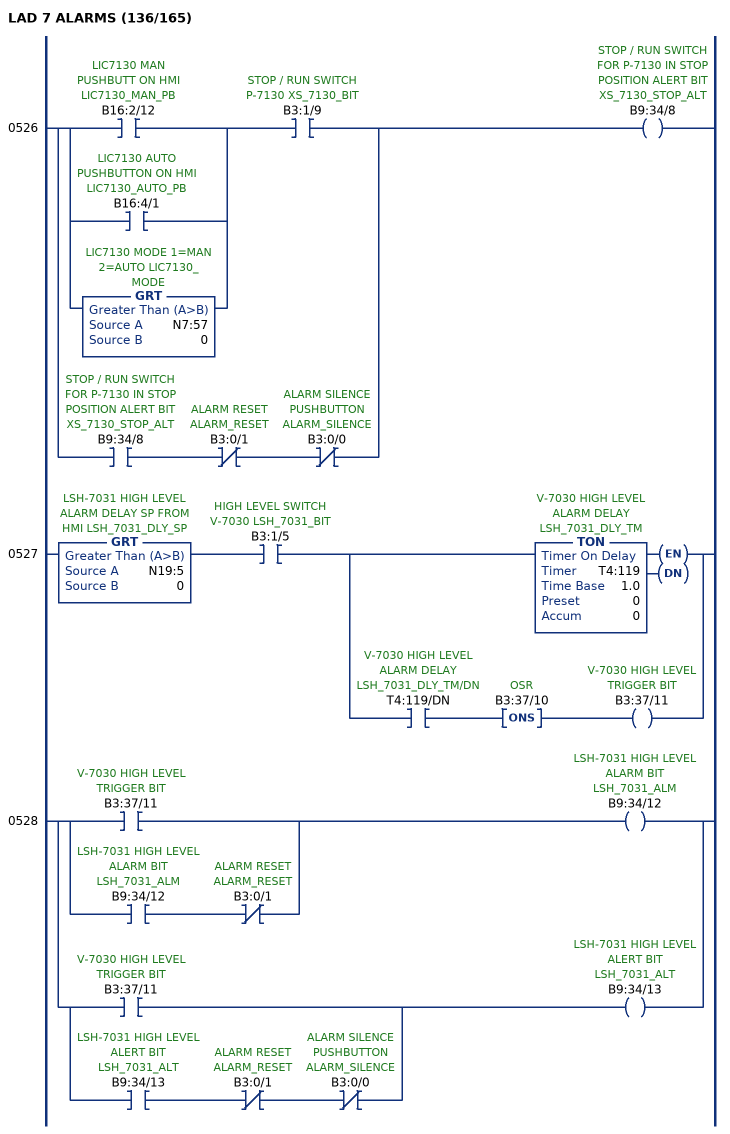
% Rung: 526 %
SOR BST BST XIC B16:2/12 NXB XIC B16:4/1 NXB GRT N7:57 0 BND XIC B3:1/9 NXB XIC B9:34/8 XIO B3:0/1 XIO B3:0/0 BND OTE B9:34/8 EOR
%   B16:2/12  LIC7130_MAN_PB  "LIC7130 MAN PUSHBUTT ON HMI" %
%   B16:4/1  LIC7130_AUTO_PB  "LIC7130 AUTO PUSHBUTTON ON HMI" %
%   N7:57  LIC7130_MODE  "LIC7130 MODE 1=MAN 2=AUTO" %
%   B3:1/9  XS_7130_BIT  "STOP / RUN SWITCH P-7130" %
%   B9:34/8  XS_7130_STOP_ALT  "STOP / RUN SWITCH FOR P-7130 IN STOP POSITION ALERT BIT" %
%   B3:0/1  ALARM_RESET  "ALARM RESET" %
%   B3:0/0  ALARM_SILENCE  "ALARM SILENCE PUSHBUTTON" %
% Rung: 527 %
SOR GRT N19:5 0 XIC B3:1/5 BST TON T4:119 1.0 0 0 NXB XIC T4:119/DN OSR B3:37/10 OTE B3:37/11 BND EOR
%   N19:5  LSH_7031_DLY_SP  "LSH-7031 HIGH LEVEL ALARM DELAY SP FROM HMI" %
%   B3:1/5  LSH_7031_BIT  "HIGH LEVEL SWITCH V-7030" %
%   T4:119  LSH_7031_DLY_TM  "V-7030 HIGH LEVEL ALARM DELAY" %
%   B3:37/10  "OSR" %
%   B3:37/11  "V-7030 HIGH LEVEL TRIGGER BIT" %
% Rung: 528 %
SOR BST BST XIC B3:37/11 NXB XIC B9:34/12 XIO B3:0/1 BND OTE B9:34/12 NXB BST XIC B3:37/11 NXB XIC B9:34/13 XIO B3:0/1 XIO B3:0/0 BND OTE B9:34/13 BND EOR
%   B3:37/11  "V-7030 HIGH LEVEL TRIGGER BIT" %
%   B9:34/12  LSH_7031_ALM  "LSH-7031 HIGH LEVEL ALARM BIT" %
%   B3:0/1  ALARM_RESET  "ALARM RESET" %
%   B9:34/13  LSH_7031_ALT  "LSH-7031 HIGH LEVEL ALERT BIT" %
%   B3:0/0  ALARM_SILENCE  "ALARM SILENCE PUSHBUTTON" %

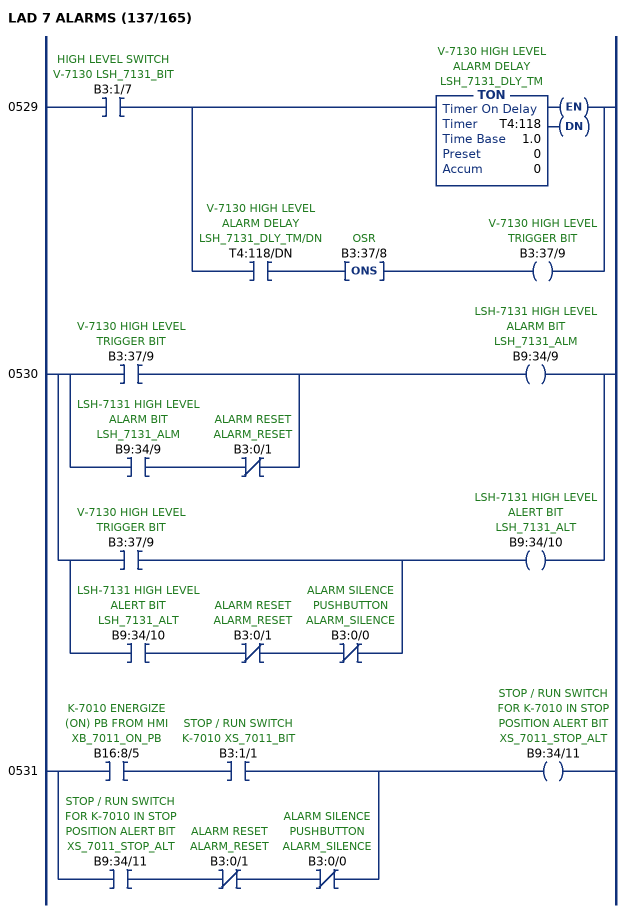
% Rung: 529 %
SOR XIC B3:1/7 BST TON T4:118 1.0 0 0 NXB XIC T4:118/DN OSR B3:37/8 OTE B3:37/9 BND EOR
%   B3:1/7  LSH_7131_BIT  "HIGH LEVEL SWITCH V-7130" %
%   T4:118  LSH_7131_DLY_TM  "V-7130 HIGH LEVEL ALARM DELAY" %
%   B3:37/8  "OSR" %
%   B3:37/9  "V-7130 HIGH LEVEL TRIGGER BIT" %
% Rung: 530 %
SOR BST BST XIC B3:37/9 NXB XIC B9:34/9 XIO B3:0/1 BND OTE B9:34/9 NXB BST XIC B3:37/9 NXB XIC B9:34/10 XIO B3:0/1 XIO B3:0/0 BND OTE B9:34/10 BND EOR
%   B3:37/9  "V-7130 HIGH LEVEL TRIGGER BIT" %
%   B9:34/9  LSH_7131_ALM  "LSH-7131 HIGH LEVEL ALARM BIT" %
%   B3:0/1  ALARM_RESET  "ALARM RESET" %
%   B9:34/10  LSH_7131_ALT  "LSH-7131 HIGH LEVEL ALERT BIT" %
%   B3:0/0  ALARM_SILENCE  "ALARM SILENCE PUSHBUTTON" %
% Rung: 531 %
SOR BST XIC B16:8/5 XIC B3:1/1 NXB XIC B9:34/11 XIO B3:0/1 XIO B3:0/0 BND OTE B9:34/11 EOR
%   B16:8/5  XB_7011_ON_PB  "K-7010 ENERGIZE (ON) PB FROM HMI" %
%   B3:1/1  XS_7011_BIT  "STOP / RUN SWITCH K-7010" %
%   B9:34/11  XS_7011_STOP_ALT  "STOP / RUN SWITCH FOR K-7010 IN STOP POSITION ALERT BIT" %
%   B3:0/1  ALARM_RESET  "ALARM RESET" %
%   B3:0/0  ALARM_SILENCE  "ALARM SILENCE PUSHBUTTON" %

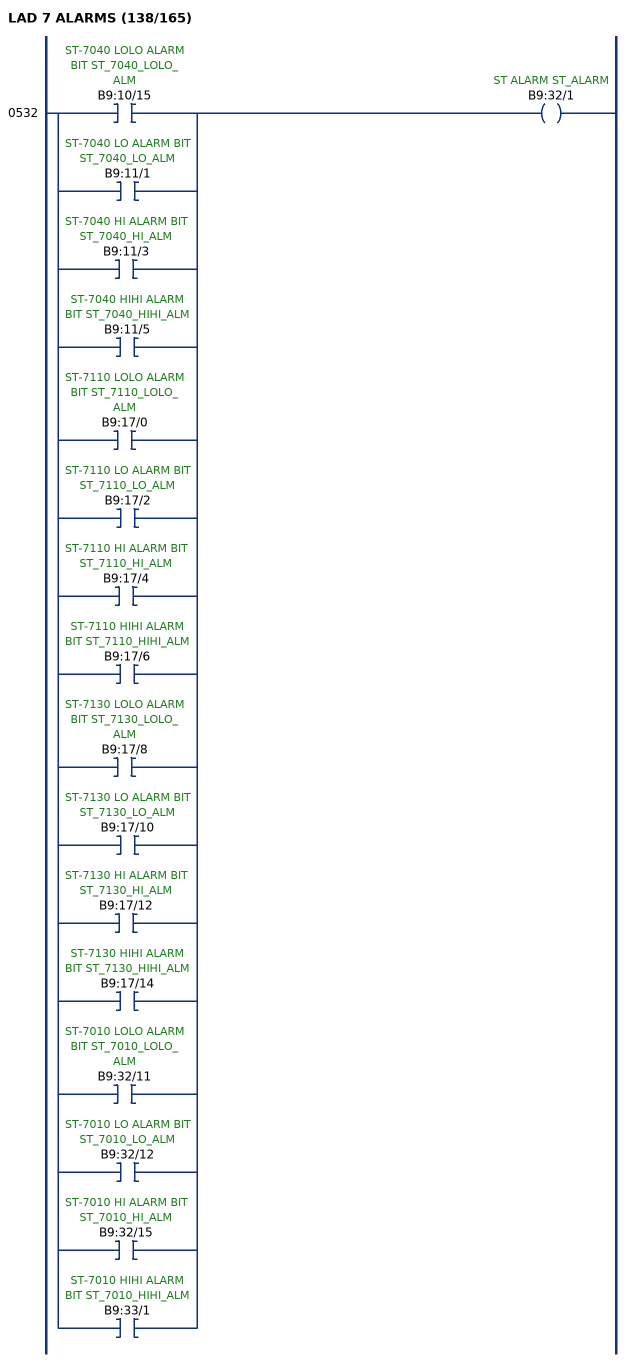
% Rung: 532 %
SOR BST XIC B9:10/15 NXB XIC B9:11/1 NXB XIC B9:11/3 NXB XIC B9:11/5 NXB XIC B9:17/0 NXB XIC B9:17/2 NXB XIC B9:17/4 NXB XIC B9:17/6 NXB XIC B9:17/8 NXB XIC B9:17/10 NXB XIC B9:17/12 NXB XIC B9:17/14 NXB XIC B9:32/11 NXB XIC B9:32/12 NXB XIC B9:32/15 NXB XIC B9:33/1 BND OTE B9:32/1 EOR
%   B9:10/15  ST_7040_LOLO_ALM  "ST-7040 LOLO ALARM BIT" %
%   B9:11/1  ST_7040_LO_ALM  "ST-7040 LO ALARM BIT" %
%   B9:11/3  ST_7040_HI_ALM  "ST-7040 HI ALARM BIT" %
%   B9:11/5  ST_7040_HIHI_ALM  "ST-7040 HIHI ALARM BIT" %
%   B9:17/0  ST_7110_LOLO_ALM  "ST-7110 LOLO ALARM BIT" %
%   B9:17/2  ST_7110_LO_ALM  "ST-7110 LO ALARM BIT" %
%   B9:17/4  ST_7110_HI_ALM  "ST-7110 HI ALARM BIT" %
%   B9:17/6  ST_7110_HIHI_ALM  "ST-7110 HIHI ALARM BIT" %
%   B9:17/8  ST_7130_LOLO_ALM  "ST-7130 LOLO ALARM BIT" %
%   B9:17/10  ST_7130_LO_ALM  "ST-7130 LO ALARM BIT" %
%   B9:17/12  ST_7130_HI_ALM  "ST-7130 HI ALARM BIT" %
%   B9:17/14  ST_7130_HIHI_ALM  "ST-7130 HIHI ALARM BIT" %
%   B9:32/11  ST_7010_LOLO_ALM  "ST-7010 LOLO ALARM BIT" %
%   B9:32/12  ST_7010_LO_ALM  "ST-7010 LO ALARM BIT" %
%   B9:32/15  ST_7010_HI_ALM  "ST-7010 HI ALARM BIT" %
%   B9:33/1  ST_7010_HIHI_ALM  "ST-7010 HIHI ALARM BIT" %
%   B9:32/1  ST_ALARM  "ST ALARM" %

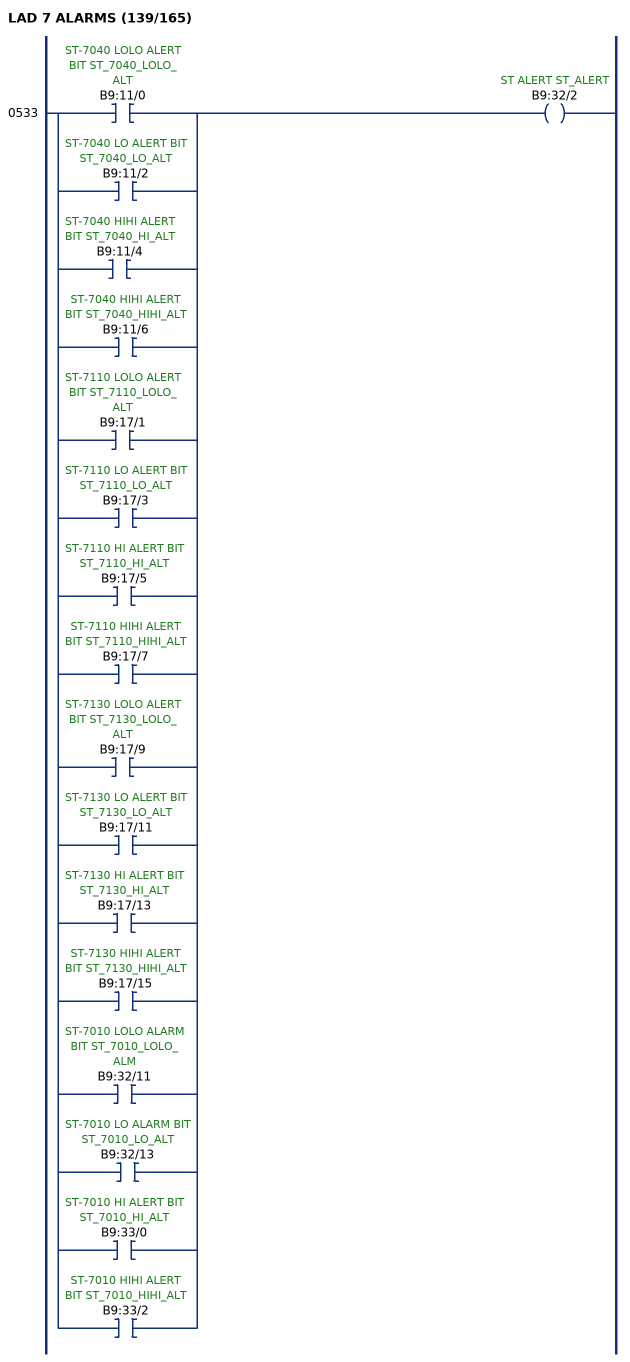
% Rung: 533 %
SOR BST XIC B9:11/0 NXB XIC B9:11/2 NXB XIC B9:11/4 NXB XIC B9:11/6 NXB XIC B9:17/1 NXB XIC B9:17/3 NXB XIC B9:17/5 NXB XIC B9:17/7 NXB XIC B9:17/9 NXB XIC B9:17/11 NXB XIC B9:17/13 NXB XIC B9:17/15 NXB XIC B9:32/11 NXB XIC B9:32/13 NXB XIC B9:33/0 NXB XIC B9:33/2 BND OTE B9:32/2 EOR
%   B9:11/0  ST_7040_LOLO_ALT  "ST-7040 LOLO ALERT BIT" %
%   B9:11/2  ST_7040_LO_ALT  "ST-7040 LO ALERT BIT" %
%   B9:11/4  ST_7040_HI_ALT  "ST-7040 HIHI ALERT BIT" %
%   B9:11/6  ST_7040_HIHI_ALT  "ST-7040 HIHI ALERT BIT" %
%   B9:17/1  ST_7110_LOLO_ALT  "ST-7110 LOLO ALERT BIT" %
%   B9:17/3  ST_7110_LO_ALT  "ST-7110 LO ALERT BIT" %
%   B9:17/5  ST_7110_HI_ALT  "ST-7110 HI ALERT BIT" %
%   B9:17/7  ST_7110_HIHI_ALT  "ST-7110 HIHI ALERT BIT" %
%   B9:17/9  ST_7130_LOLO_ALT  "ST-7130 LOLO ALERT BIT" %
%   B9:17/11  ST_7130_LO_ALT  "ST-7130 LO ALERT BIT" %
%   B9:17/13  ST_7130_HI_ALT  "ST-7130 HI ALERT BIT" %
%   B9:17/15  ST_7130_HIHI_ALT  "ST-7130 HIHI ALERT BIT" %
%   B9:32/11  ST_7010_LOLO_ALM  "ST-7010 LOLO ALARM BIT" %
%   B9:32/13  ST_7010_LO_ALT  "ST-7010 LO ALARM BIT" %
%   B9:33/0  ST_7010_HI_ALT  "ST-7010 HI ALERT BIT" %
%   B9:33/2  ST_7010_HIHI_ALT  "ST-7010 HIHI ALERT BIT" %
%   B9:32/2  ST_ALERT  "ST ALERT" %

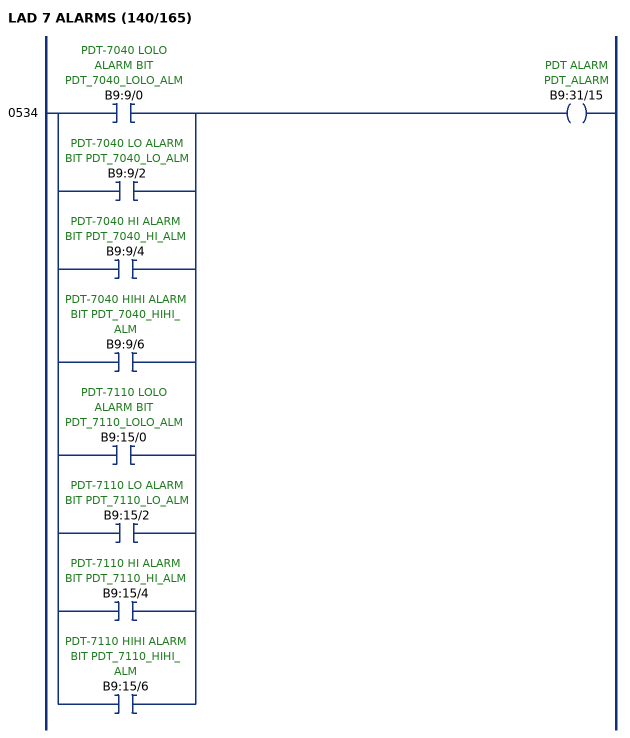
% Rung: 534 %
SOR BST XIC B9:9/0 NXB XIC B9:9/2 NXB XIC B9:9/4 NXB XIC B9:9/6 NXB XIC B9:15/0 NXB XIC B9:15/2 NXB XIC B9:15/4 NXB XIC B9:15/6 BND OTE B9:31/15 EOR
%   B9:9/0  PDT_7040_LOLO_ALM  "PDT-7040 LOLO ALARM BIT" %
%   B9:9/2  PDT_7040_LO_ALM  "PDT-7040 LO ALARM BIT" %
%   B9:9/4  PDT_7040_HI_ALM  "PDT-7040 HI ALARM BIT" %
%   B9:9/6  PDT_7040_HIHI_ALM  "PDT-7040 HIHI ALARM BIT" %
%   B9:15/0  PDT_7110_LOLO_ALM  "PDT-7110 LOLO ALARM BIT" %
%   B9:15/2  PDT_7110_LO_ALM  "PDT-7110 LO ALARM BIT" %
%   B9:15/4  PDT_7110_HI_ALM  "PDT-7110 HI ALARM BIT" %
%   B9:15/6  PDT_7110_HIHI_ALM  "PDT-7110 HIHI ALARM BIT" %
%   B9:31/15  PDT_ALARM  "PDT ALARM" %

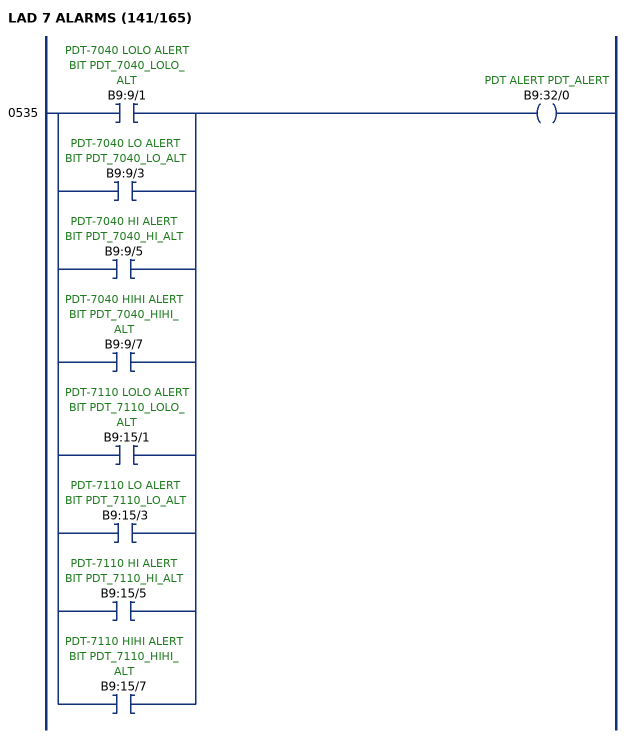
% Rung: 535 %
SOR BST XIC B9:9/1 NXB XIC B9:9/3 NXB XIC B9:9/5 NXB XIC B9:9/7 NXB XIC B9:15/1 NXB XIC B9:15/3 NXB XIC B9:15/5 NXB XIC B9:15/7 BND OTE B9:32/0 EOR
%   B9:9/1  PDT_7040_LOLO_ALT  "PDT-7040 LOLO ALERT BIT" %
%   B9:9/3  PDT_7040_LO_ALT  "PDT-7040 LO ALERT BIT" %
%   B9:9/5  PDT_7040_HI_ALT  "PDT-7040 HI ALERT BIT" %
%   B9:9/7  PDT_7040_HIHI_ALT  "PDT-7040 HIHI ALERT BIT" %
%   B9:15/1  PDT_7110_LOLO_ALT  "PDT-7110 LOLO ALERT BIT" %
%   B9:15/3  PDT_7110_LO_ALT  "PDT-7110 LO ALERT BIT" %
%   B9:15/5  PDT_7110_HI_ALT  "PDT-7110 HI ALERT BIT" %
%   B9:15/7  PDT_7110_HIHI_ALT  "PDT-7110 HIHI ALERT BIT" %
%   B9:32/0  PDT_ALERT  "PDT ALERT" %

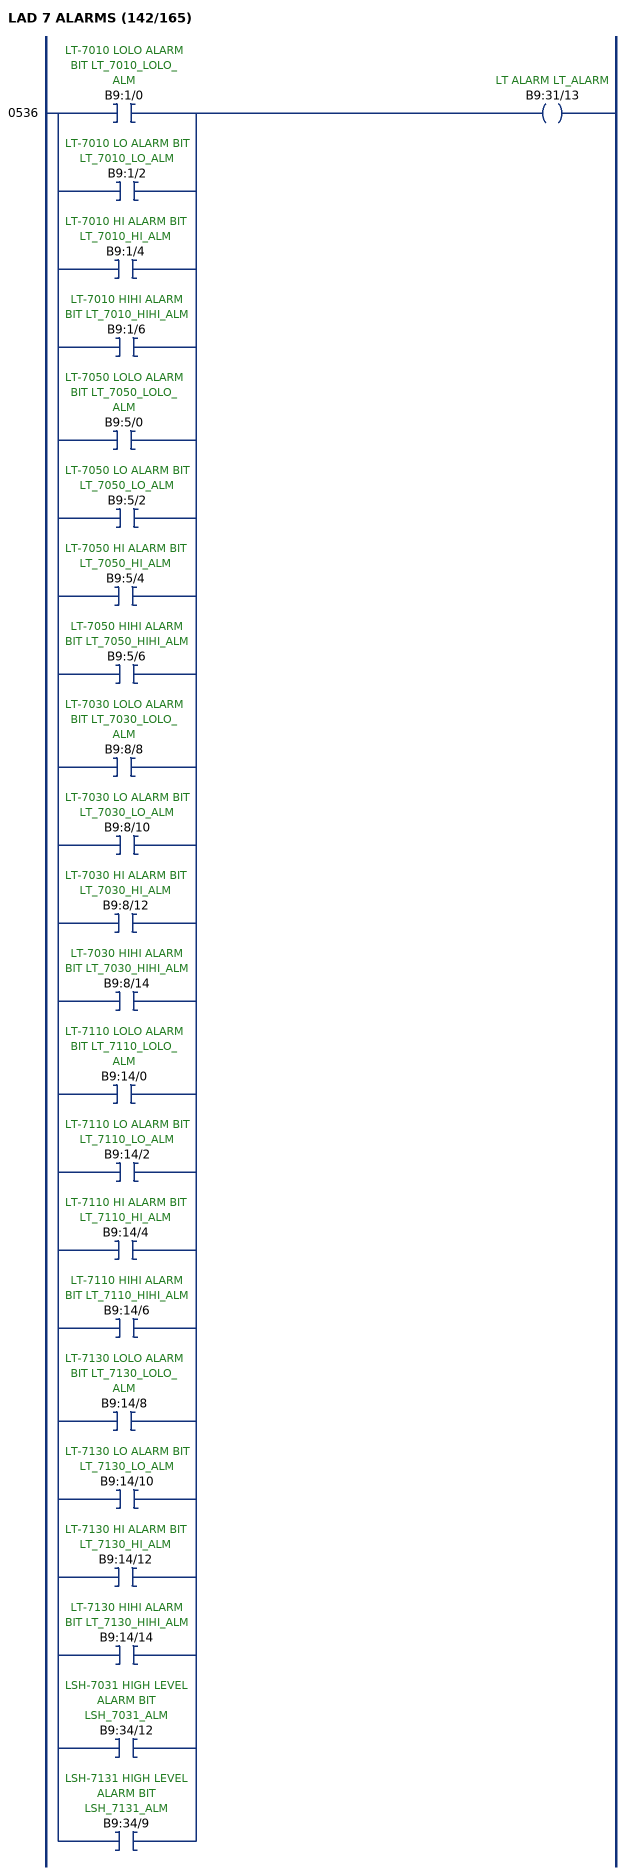
% Rung: 536 %
SOR BST XIC B9:1/0 NXB XIC B9:1/2 NXB XIC B9:1/4 NXB XIC B9:1/6 NXB XIC B9:5/0 NXB XIC B9:5/2 NXB XIC B9:5/4 NXB XIC B9:5/6 NXB XIC B9:8/8 NXB XIC B9:8/10 NXB XIC B9:8/12 NXB XIC B9:8/14 NXB XIC B9:14/0 NXB XIC B9:14/2 NXB XIC B9:14/4 NXB XIC B9:14/6 NXB XIC B9:14/8 NXB XIC B9:14/10 NXB XIC B9:14/12 NXB XIC B9:14/14 NXB XIC B9:34/12 NXB XIC B9:34/9 BND OTE B9:31/13 EOR
%   B9:1/0  LT_7010_LOLO_ALM  "LT-7010 LOLO ALARM BIT" %
%   B9:1/2  LT_7010_LO_ALM  "LT-7010 LO ALARM BIT" %
%   B9:1/4  LT_7010_HI_ALM  "LT-7010 HI ALARM BIT" %
%   B9:1/6  LT_7010_HIHI_ALM  "LT-7010 HIHI ALARM BIT" %
%   B9:5/0  LT_7050_LOLO_ALM  "LT-7050 LOLO ALARM BIT" %
%   B9:5/2  LT_7050_LO_ALM  "LT-7050 LO ALARM BIT" %
%   B9:5/4  LT_7050_HI_ALM  "LT-7050 HI ALARM BIT" %
%   B9:5/6  LT_7050_HIHI_ALM  "LT-7050 HIHI ALARM BIT" %
%   B9:8/8  LT_7030_LOLO_ALM  "LT-7030 LOLO ALARM BIT" %
%   B9:8/10  LT_7030_LO_ALM  "LT-7030 LO ALARM BIT" %
%   B9:8/12  LT_7030_HI_ALM  "LT-7030 HI ALARM BIT" %
%   B9:8/14  LT_7030_HIHI_ALM  "LT-7030 HIHI ALARM BIT" %
%   B9:14/0  LT_7110_LOLO_ALM  "LT-7110 LOLO ALARM BIT" %
%   B9:14/2  LT_7110_LO_ALM  "LT-7110 LO ALARM BIT" %
%   B9:14/4  LT_7110_HI_ALM  "LT-7110 HI ALARM BIT" %
%   B9:14/6  LT_7110_HIHI_ALM  "LT-7110 HIHI ALARM BIT" %
%   B9:14/8  LT_7130_LOLO_ALM  "LT-7130 LOLO ALARM BIT" %
%   B9:14/10  LT_7130_LO_ALM  "LT-7130 LO ALARM BIT" %
%   B9:14/12  LT_7130_HI_ALM  "LT-7130 HI ALARM BIT" %
%   B9:14/14  LT_7130_HIHI_ALM  "LT-7130 HIHI ALARM BIT" %
%   B9:34/12  LSH_7031_ALM  "LSH-7031 HIGH LEVEL ALARM BIT" %
%   B9:34/9  LSH_7131_ALM  "LSH-7131 HIGH LEVEL ALARM BIT" %
%   B9:31/13  LT_ALARM  "LT ALARM" %

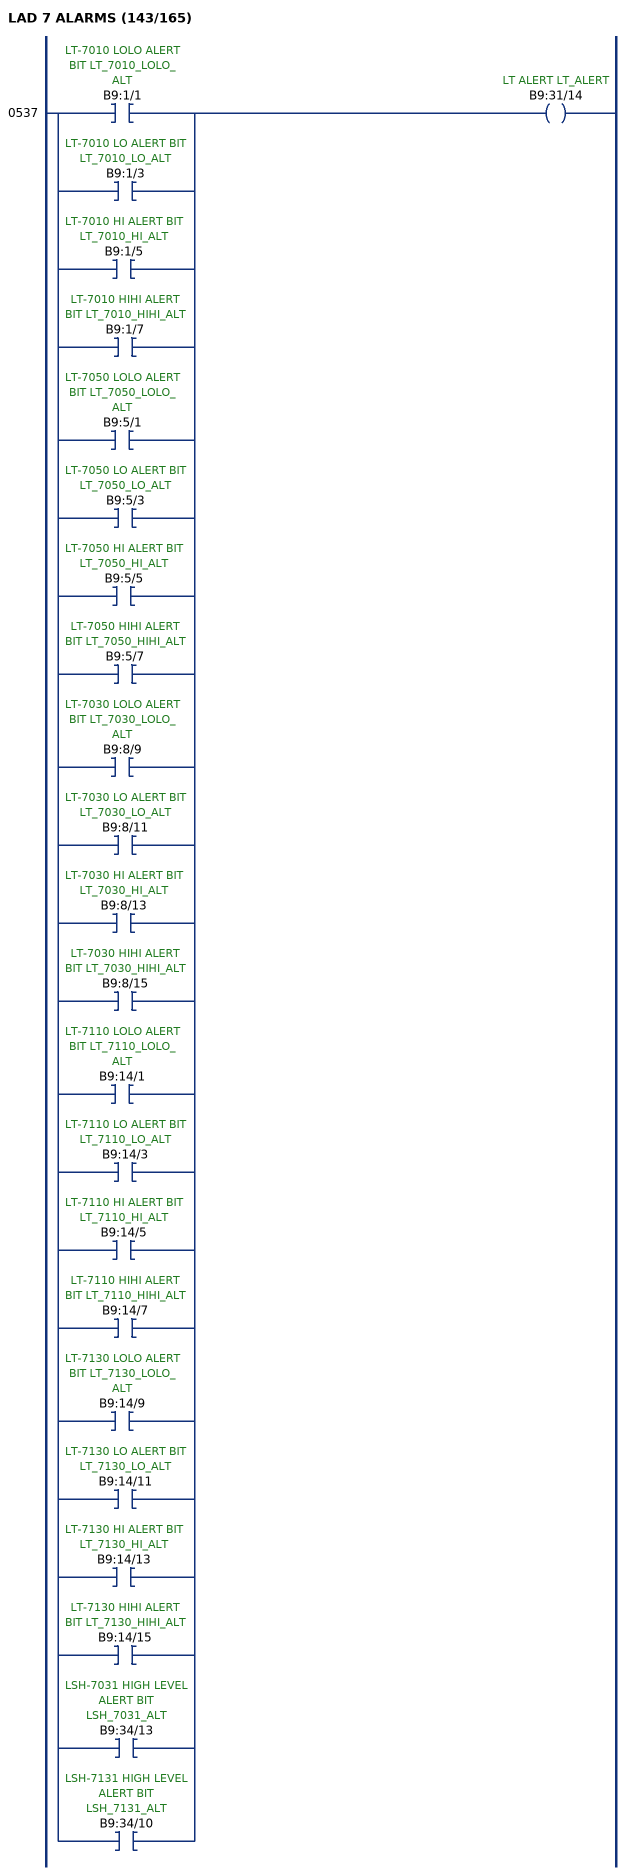
% Rung: 537 %
SOR BST XIC B9:1/1 NXB XIC B9:1/3 NXB XIC B9:1/5 NXB XIC B9:1/7 NXB XIC B9:5/1 NXB XIC B9:5/3 NXB XIC B9:5/5 NXB XIC B9:5/7 NXB XIC B9:8/9 NXB XIC B9:8/11 NXB XIC B9:8/13 NXB XIC B9:8/15 NXB XIC B9:14/1 NXB XIC B9:14/3 NXB XIC B9:14/5 NXB XIC B9:14/7 NXB XIC B9:14/9 NXB XIC B9:14/11 NXB XIC B9:14/13 NXB XIC B9:14/15 NXB XIC B9:34/13 NXB XIC B9:34/10 BND OTE B9:31/14 EOR
%   B9:1/1  LT_7010_LOLO_ALT  "LT-7010 LOLO ALERT BIT" %
%   B9:1/3  LT_7010_LO_ALT  "LT-7010 LO ALERT BIT" %
%   B9:1/5  LT_7010_HI_ALT  "LT-7010 HI ALERT BIT" %
%   B9:1/7  LT_7010_HIHI_ALT  "LT-7010 HIHI ALERT BIT" %
%   B9:5/1  LT_7050_LOLO_ALT  "LT-7050 LOLO ALERT BIT" %
%   B9:5/3  LT_7050_LO_ALT  "LT-7050 LO ALERT BIT" %
%   B9:5/5  LT_7050_HI_ALT  "LT-7050 HI ALERT BIT" %
%   B9:5/7  LT_7050_HIHI_ALT  "LT-7050 HIHI ALERT BIT" %
%   B9:8/9  LT_7030_LOLO_ALT  "LT-7030 LOLO ALERT BIT" %
%   B9:8/11  LT_7030_LO_ALT  "LT-7030 LO ALERT BIT" %
%   B9:8/13  LT_7030_HI_ALT  "LT-7030 HI ALERT BIT" %
%   B9:8/15  LT_7030_HIHI_ALT  "LT-7030 HIHI ALERT BIT" %
%   B9:14/1  LT_7110_LOLO_ALT  "LT-7110 LOLO ALERT BIT" %
%   B9:14/3  LT_7110_LO_ALT  "LT-7110 LO ALERT BIT" %
%   B9:14/5  LT_7110_HI_ALT  "LT-7110 HI ALERT BIT" %
%   B9:14/7  LT_7110_HIHI_ALT  "LT-7110 HIHI ALERT BIT" %
%   B9:14/9  LT_7130_LOLO_ALT  "LT-7130 LOLO ALERT BIT" %
%   B9:14/11  LT_7130_LO_ALT  "LT-7130 LO ALERT BIT" %
%   B9:14/13  LT_7130_HI_ALT  "LT-7130 HI ALERT BIT" %
%   B9:14/15  LT_7130_HIHI_ALT  "LT-7130 HIHI ALERT BIT" %
%   B9:34/13  LSH_7031_ALT  "LSH-7031 HIGH LEVEL ALERT BIT" %
%   B9:34/10  LSH_7131_ALT  "LSH-7131 HIGH LEVEL ALERT BIT" %
%   B9:31/14  LT_ALERT  "LT ALERT" %

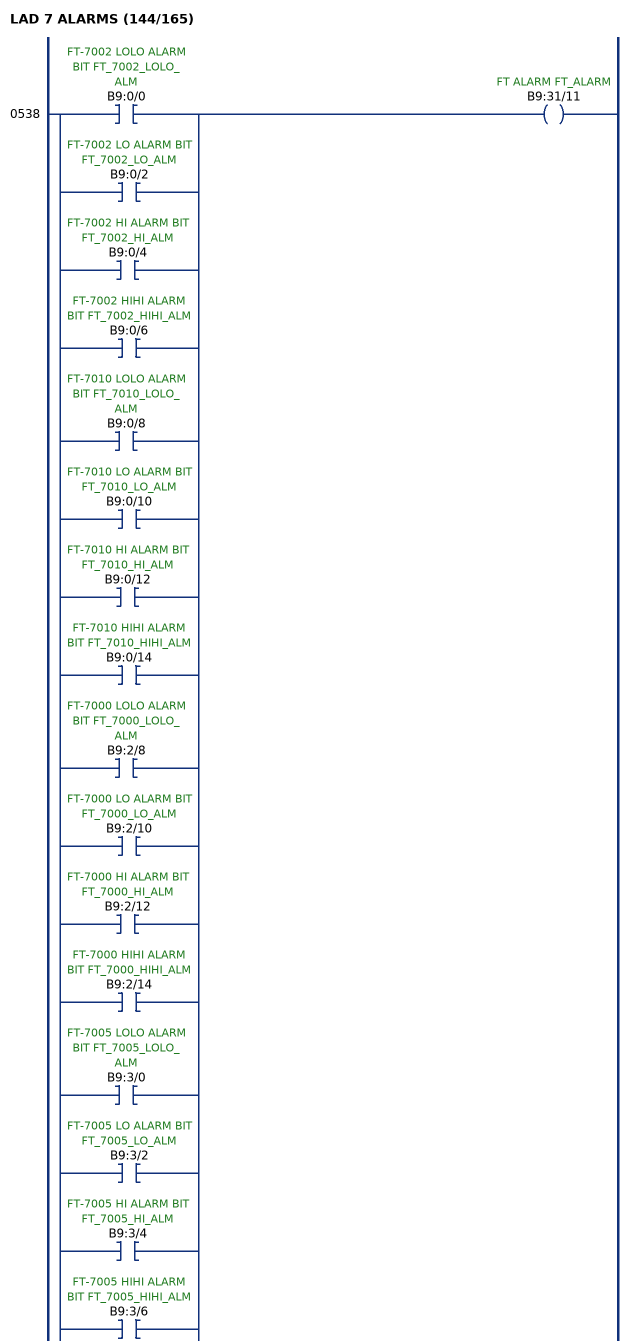

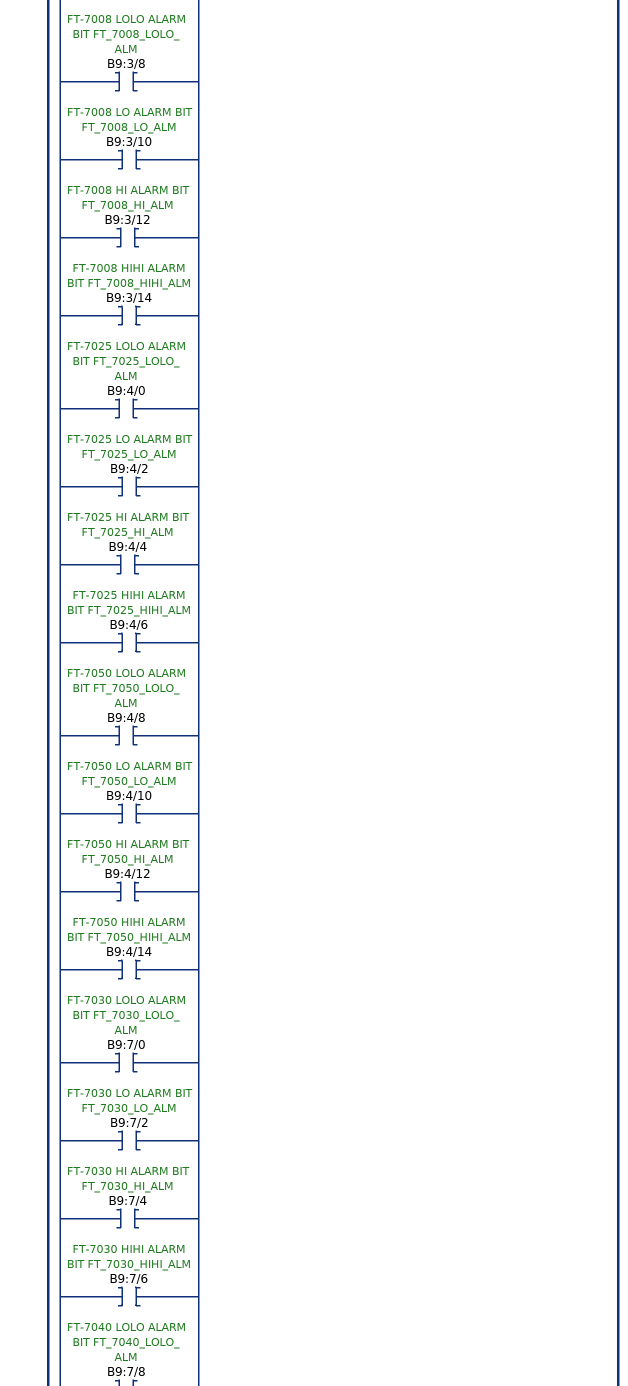

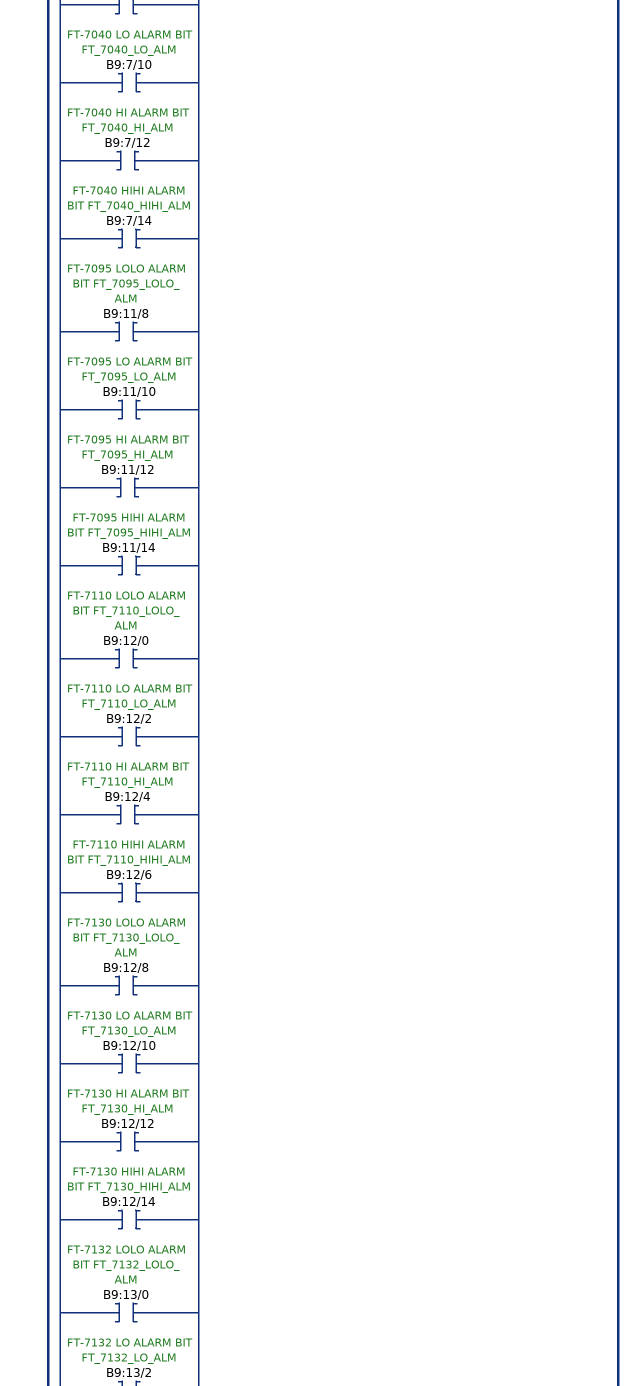

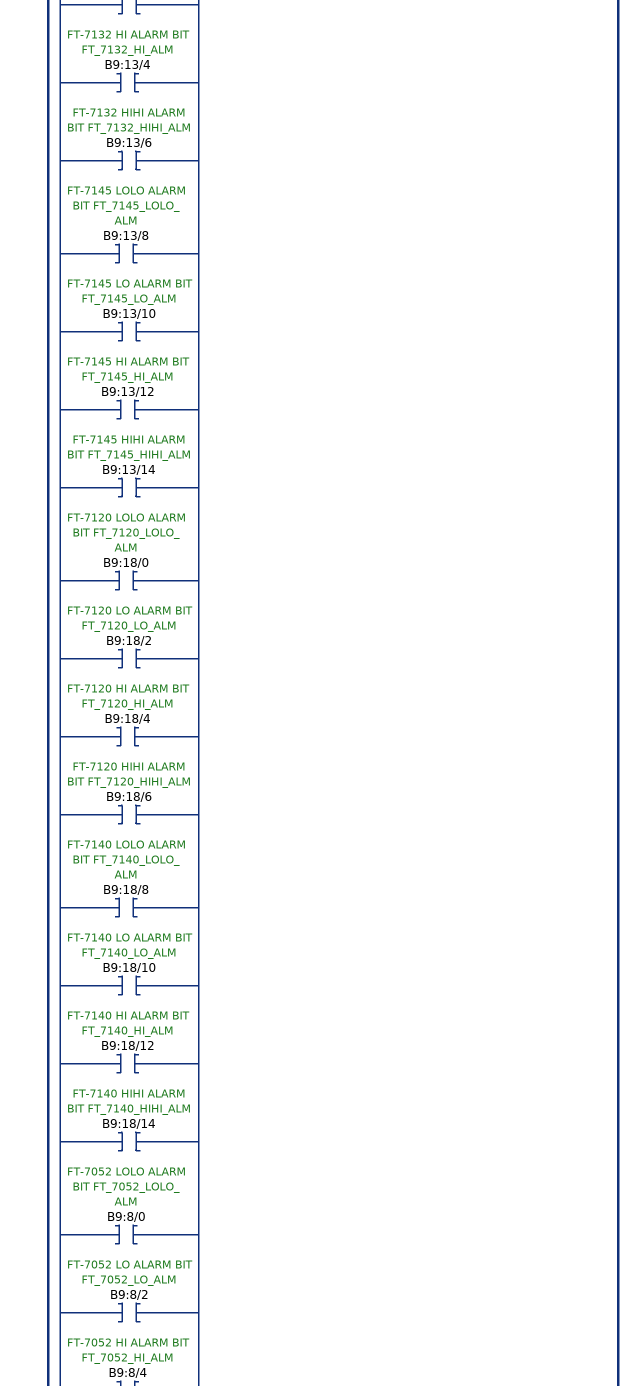

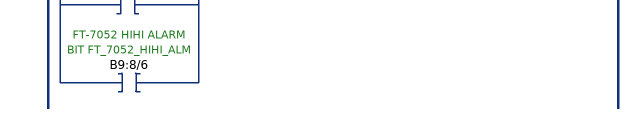
% Rung: 538 %
SOR BST XIC B9:0/0 NXB XIC B9:0/2 NXB XIC B9:0/4 NXB XIC B9:0/6 NXB XIC B9:0/8 NXB XIC B9:0/10 NXB XIC B9:0/12 NXB XIC B9:0/14 NXB XIC B9:2/8 NXB XIC B9:2/10 NXB XIC B9:2/12 NXB XIC B9:2/14 NXB XIC B9:3/0 NXB XIC B9:3/2 NXB XIC B9:3/4 NXB XIC B9:3/6 NXB XIC B9:3/8 NXB XIC B9:3/10 NXB XIC B9:3/12 NXB XIC B9:3/14 NXB XIC B9:4/0 NXB XIC B9:4/2 NXB XIC B9:4/4 NXB XIC B9:4/6 NXB XIC B9:4/8 NXB XIC B9:4/10 NXB XIC B9:4/12 NXB XIC B9:4/14 NXB XIC B9:7/0 NXB XIC B9:7/2 NXB XIC B9:7/4 NXB XIC B9:7/6 NXB XIC B9:7/8 NXB XIC B9:7/10 NXB XIC B9:7/12 NXB XIC B9:7/14 NXB XIC B9:11/8 NXB XIC B9:11/10 NXB XIC B9:11/12 NXB XIC B9:11/14 NXB XIC B9:12/0 NXB XIC B9:12/2 NXB XIC B9:12/4 NXB XIC B9:12/6 NXB XIC B9:12/8 NXB XIC B9:12/10 NXB XIC B9:12/12 NXB XIC B9:12/14 NXB XIC B9:13/0 NXB XIC B9:13/2 NXB XIC B9:13/4 NXB XIC B9:13/6 NXB XIC B9:13/8 NXB XIC B9:13/10 NXB XIC B9:13/12 NXB XIC B9:13/14 NXB XIC B9:18/0 NXB XIC B9:18/2 NXB XIC B9:18/4 NXB XIC B9:18/6 NXB XIC B9:18/8 NXB XIC B9:18/10 NXB XIC B9:18/12 NXB XIC B9:18/14 NXB XIC B9:8/0 NXB XIC B9:8/2 NXB XIC B9:8/4 NXB XIC B9:8/6 BND OTE B9:31/11 EOR
%   B9:0/0  FT_7002_LOLO_ALM  "FT-7002 LOLO ALARM BIT" %
%   B9:0/2  FT_7002_LO_ALM  "FT-7002 LO ALARM BIT" %
%   B9:0/4  FT_7002_HI_ALM  "FT-7002 HI ALARM BIT" %
%   B9:0/6  FT_7002_HIHI_ALM  "FT-7002 HIHI ALARM BIT" %
%   B9:0/8  FT_7010_LOLO_ALM  "FT-7010 LOLO ALARM BIT" %
%   B9:0/10  FT_7010_LO_ALM  "FT-7010 LO ALARM BIT" %
%   B9:0/12  FT_7010_HI_ALM  "FT-7010 HI ALARM BIT" %
%   B9:0/14  FT_7010_HIHI_ALM  "FT-7010 HIHI ALARM BIT" %
%   B9:2/8  FT_7000_LOLO_ALM  "FT-7000 LOLO ALARM BIT" %
%   B9:2/10  FT_7000_LO_ALM  "FT-7000 LO ALARM BIT" %
%   B9:2/12  FT_7000_HI_ALM  "FT-7000 HI ALARM BIT" %
%   B9:2/14  FT_7000_HIHI_ALM  "FT-7000 HIHI ALARM BIT" %
%   B9:3/0  FT_7005_LOLO_ALM  "FT-7005 LOLO ALARM BIT" %
%   B9:3/2  FT_7005_LO_ALM  "FT-7005 LO ALARM BIT" %
%   B9:3/4  FT_7005_HI_ALM  "FT-7005 HI ALARM BIT" %
%   B9:3/6  FT_7005_HIHI_ALM  "FT-7005 HIHI ALARM BIT" %
%   B9:3/8  FT_7008_LOLO_ALM  "FT-7008 LOLO ALARM BIT" %
%   B9:3/10  FT_7008_LO_ALM  "FT-7008 LO ALARM BIT" %
%   B9:3/12  FT_7008_HI_ALM  "FT-7008 HI ALARM BIT" %
%   B9:3/14  FT_7008_HIHI_ALM  "FT-7008 HIHI ALARM BIT" %
%   B9:4/0  FT_7025_LOLO_ALM  "FT-7025 LOLO ALARM BIT" %
%   B9:4/2  FT_7025_LO_ALM  "FT-7025 LO ALARM BIT" %
%   B9:4/4  FT_7025_HI_ALM  "FT-7025 HI ALARM BIT" %
%   B9:4/6  FT_7025_HIHI_ALM  "FT-7025 HIHI ALARM BIT" %
%   B9:4/8  FT_7050_LOLO_ALM  "FT-7050 LOLO ALARM BIT" %
%   B9:4/10  FT_7050_LO_ALM  "FT-7050 LO ALARM BIT" %
%   B9:4/12  FT_7050_HI_ALM  "FT-7050 HI ALARM BIT" %
%   B9:4/14  FT_7050_HIHI_ALM  "FT-7050 HIHI ALARM BIT" %
%   B9:7/0  FT_7030_LOLO_ALM  "FT-7030 LOLO ALARM BIT" %
%   B9:7/2  FT_7030_LO_ALM  "FT-7030 LO ALARM BIT" %
%   B9:7/4  FT_7030_HI_ALM  "FT-7030 HI ALARM BIT" %
%   B9:7/6  FT_7030_HIHI_ALM  "FT-7030 HIHI ALARM BIT" %
%   B9:7/8  FT_7040_LOLO_ALM  "FT-7040 LOLO ALARM BIT" %
%   B9:7/10  FT_7040_LO_ALM  "FT-7040 LO ALARM BIT" %
%   B9:7/12  FT_7040_HI_ALM  "FT-7040 HI ALARM BIT" %
%   B9:7/14  FT_7040_HIHI_ALM  "FT-7040 HIHI ALARM BIT" %
%   B9:11/8  FT_7095_LOLO_ALM  "FT-7095 LOLO ALARM BIT" %
%   B9:11/10  FT_7095_LO_ALM  "FT-7095 LO ALARM BIT" %
%   B9:11/12  FT_7095_HI_ALM  "FT-7095 HI ALARM BIT" %
%   B9:11/14  FT_7095_HIHI_ALM  "FT-7095 HIHI ALARM BIT" %
%   B9:12/0  FT_7110_LOLO_ALM  "FT-7110 LOLO ALARM BIT" %
%   B9:12/2  FT_7110_LO_ALM  "FT-7110 LO ALARM BIT" %
%   B9:12/4  FT_7110_HI_ALM  "FT-7110 HI ALARM BIT" %
%   B9:12/6  FT_7110_HIHI_ALM  "FT-7110 HIHI ALARM BIT" %
%   B9:12/8  FT_7130_LOLO_ALM  "FT-7130 LOLO ALARM BIT" %
%   B9:12/10  FT_7130_LO_ALM  "FT-7130 LO ALARM BIT" %
%   B9:12/12  FT_7130_HI_ALM  "FT-7130 HI ALARM BIT" %
%   B9:12/14  FT_7130_HIHI_ALM  "FT-7130 HIHI ALARM BIT" %
%   B9:13/0  FT_7132_LOLO_ALM  "FT-7132 LOLO ALARM BIT" %
%   B9:13/2  FT_7132_LO_ALM  "FT-7132 LO ALARM BIT" %
%   B9:13/4  FT_7132_HI_ALM  "FT-7132 HI ALARM BIT" %
%   B9:13/6  FT_7132_HIHI_ALM  "FT-7132 HIHI ALARM BIT" %
%   B9:13/8  FT_7145_LOLO_ALM  "FT-7145 LOLO ALARM BIT" %
%   B9:13/10  FT_7145_LO_ALM  "FT-7145 LO ALARM BIT" %
%   B9:13/12  FT_7145_HI_ALM  "FT-7145 HI ALARM BIT" %
%   B9:13/14  FT_7145_HIHI_ALM  "FT-7145 HIHI ALARM BIT" %
%   B9:18/0  FT_7120_LOLO_ALM  "FT-7120 LOLO ALARM BIT" %
%   B9:18/2  FT_7120_LO_ALM  "FT-7120 LO ALARM BIT" %
%   B9:18/4  FT_7120_HI_ALM  "FT-7120 HI ALARM BIT" %
%   B9:18/6  FT_7120_HIHI_ALM  "FT-7120 HIHI ALARM BIT" %
%   B9:18/8  FT_7140_LOLO_ALM  "FT-7140 LOLO ALARM BIT" %
%   B9:18/10  FT_7140_LO_ALM  "FT-7140 LO ALARM BIT" %
%   B9:18/12  FT_7140_HI_ALM  "FT-7140 HI ALARM BIT" %
%   B9:18/14  FT_7140_HIHI_ALM  "FT-7140 HIHI ALARM BIT" %
%   B9:8/0  FT_7052_LOLO_ALM  "FT-7052 LOLO ALARM BIT" %
%   B9:8/2  FT_7052_LO_ALM  "FT-7052 LO ALARM BIT" %
%   B9:8/4  FT_7052_HI_ALM  "FT-7052 HI ALARM BIT" %
%   B9:8/6  FT_7052_HIHI_ALM  "FT-7052 HIHI ALARM BIT" %
%   B9:31/11  FT_ALARM  "FT ALARM" %

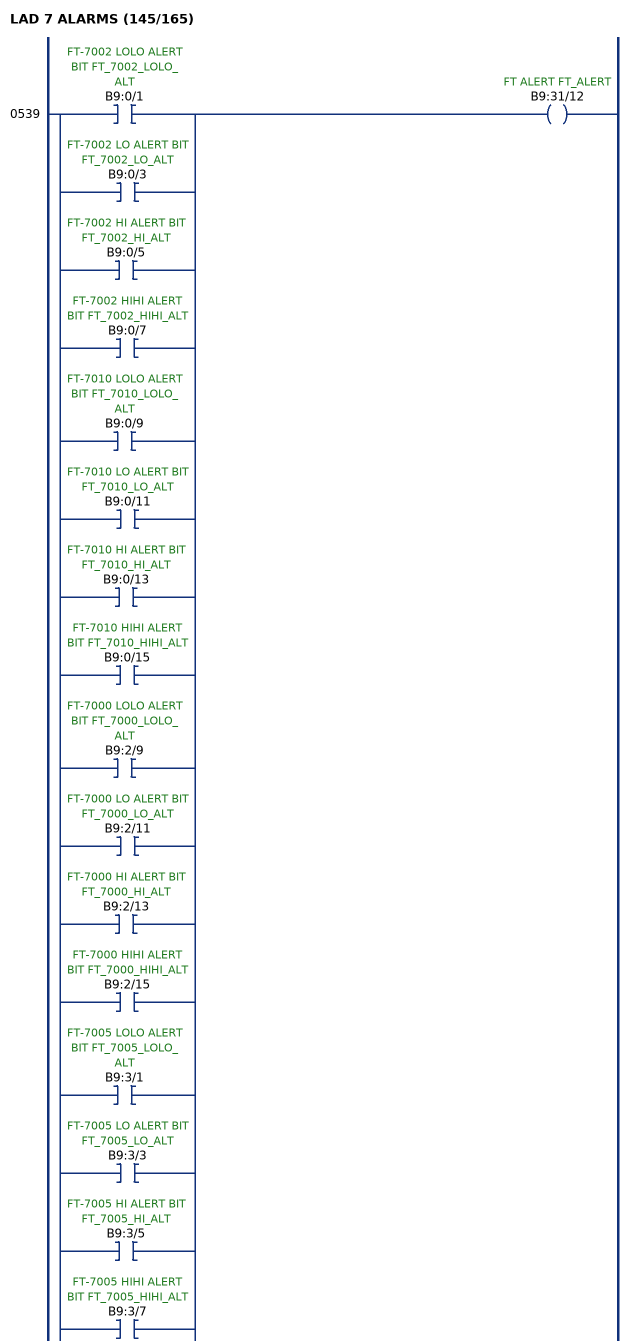

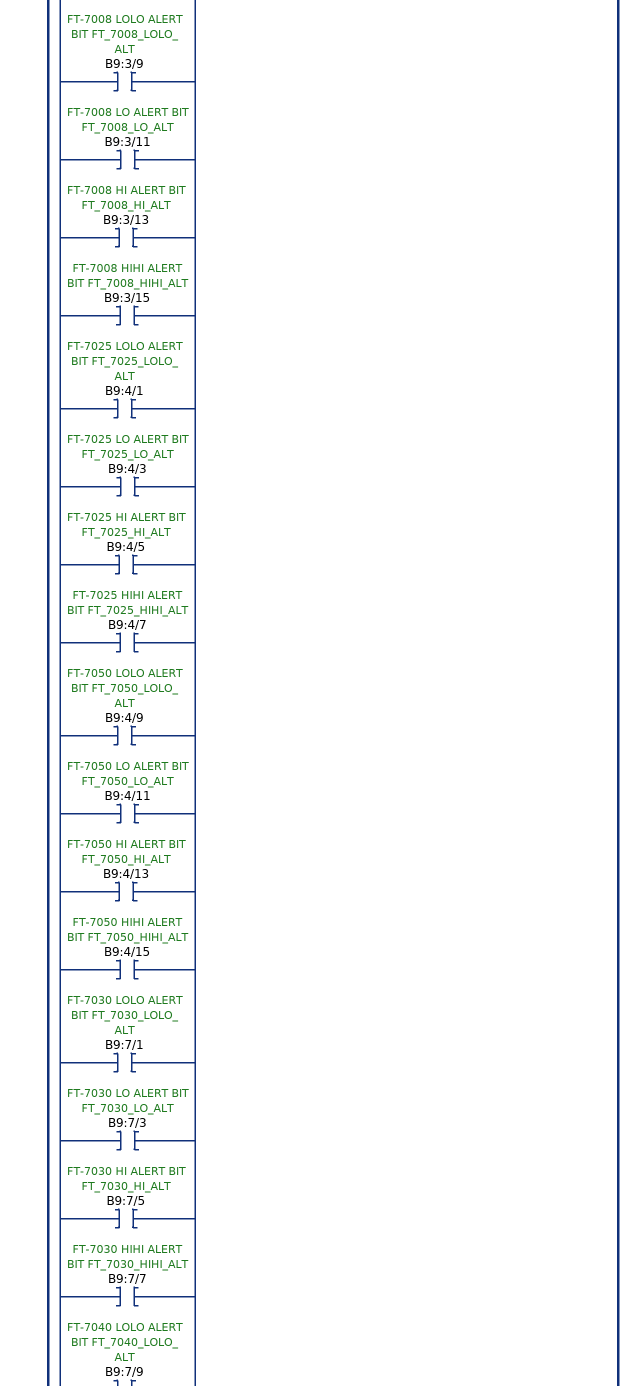

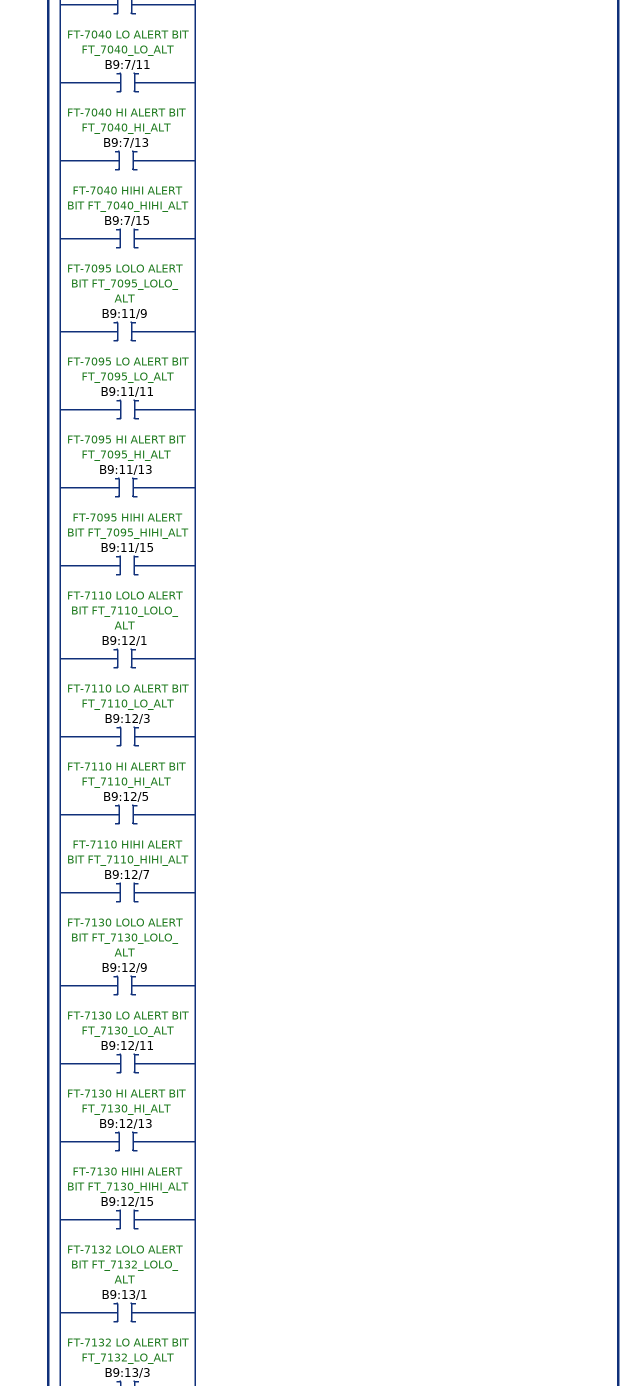

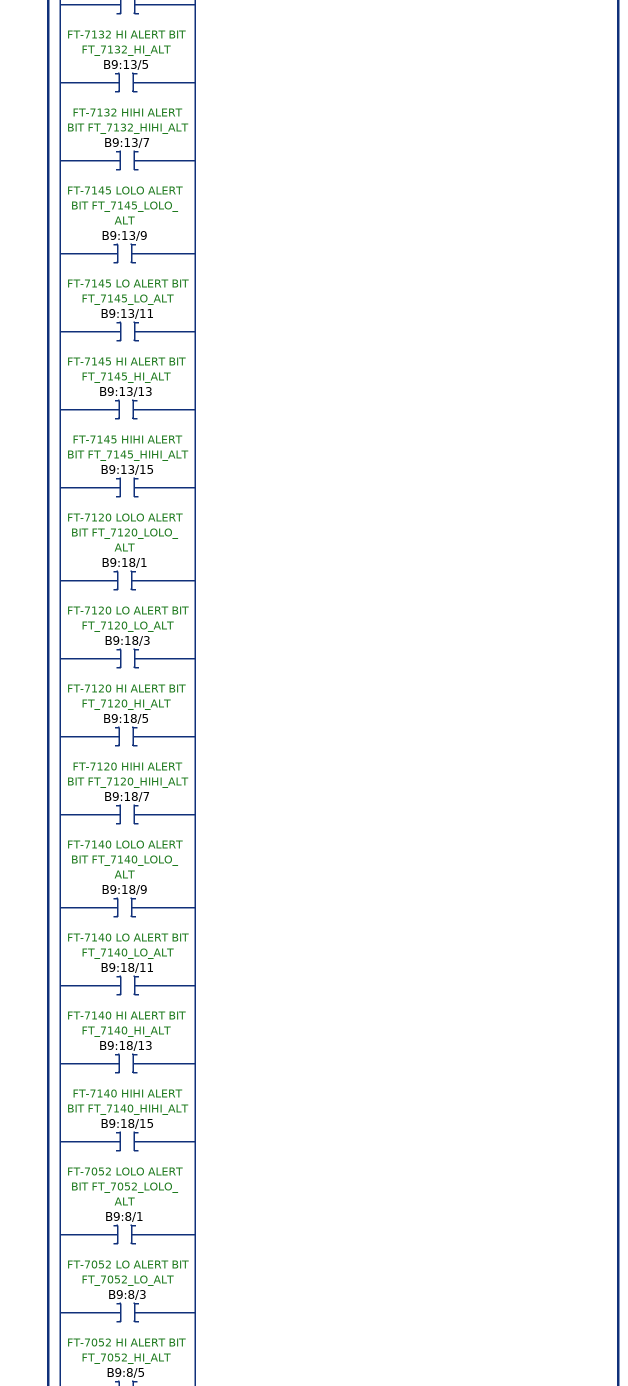

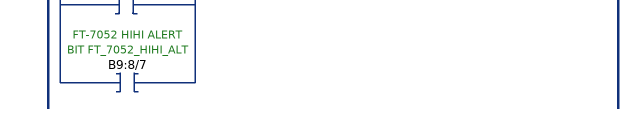
% Rung: 539 %
SOR BST XIC B9:0/1 NXB XIC B9:0/3 NXB XIC B9:0/5 NXB XIC B9:0/7 NXB XIC B9:0/9 NXB XIC B9:0/11 NXB XIC B9:0/13 NXB XIC B9:0/15 NXB XIC B9:2/9 NXB XIC B9:2/11 NXB XIC B9:2/13 NXB XIC B9:2/15 NXB XIC B9:3/1 NXB XIC B9:3/3 NXB XIC B9:3/5 NXB XIC B9:3/7 NXB XIC B9:3/9 NXB XIC B9:3/11 NXB XIC B9:3/13 NXB XIC B9:3/15 NXB XIC B9:4/1 NXB XIC B9:4/3 NXB XIC B9:4/5 NXB XIC B9:4/7 NXB XIC B9:4/9 NXB XIC B9:4/11 NXB XIC B9:4/13 NXB XIC B9:4/15 NXB XIC B9:7/1 NXB XIC B9:7/3 NXB XIC B9:7/5 NXB XIC B9:7/7 NXB XIC B9:7/9 NXB XIC B9:7/11 NXB XIC B9:7/13 NXB XIC B9:7/15 NXB XIC B9:11/9 NXB XIC B9:11/11 NXB XIC B9:11/13 NXB XIC B9:11/15 NXB XIC B9:12/1 NXB XIC B9:12/3 NXB XIC B9:12/5 NXB XIC B9:12/7 NXB XIC B9:12/9 NXB XIC B9:12/11 NXB XIC B9:12/13 NXB XIC B9:12/15 NXB XIC B9:13/1 NXB XIC B9:13/3 NXB XIC B9:13/5 NXB XIC B9:13/7 NXB XIC B9:13/9 NXB XIC B9:13/11 NXB XIC B9:13/13 NXB XIC B9:13/15 NXB XIC B9:18/1 NXB XIC B9:18/3 NXB XIC B9:18/5 NXB XIC B9:18/7 NXB XIC B9:18/9 NXB XIC B9:18/11 NXB XIC B9:18/13 NXB XIC B9:18/15 NXB XIC B9:8/1 NXB XIC B9:8/3 NXB XIC B9:8/5 NXB XIC B9:8/7 BND OTE B9:31/12 EOR
%   B9:0/1  FT_7002_LOLO_ALT  "FT-7002 LOLO ALERT BIT" %
%   B9:0/3  FT_7002_LO_ALT  "FT-7002 LO ALERT BIT" %
%   B9:0/5  FT_7002_HI_ALT  "FT-7002 HI ALERT BIT" %
%   B9:0/7  FT_7002_HIHI_ALT  "FT-7002 HIHI ALERT BIT" %
%   B9:0/9  FT_7010_LOLO_ALT  "FT-7010 LOLO ALERT BIT" %
%   B9:0/11  FT_7010_LO_ALT  "FT-7010 LO ALERT BIT" %
%   B9:0/13  FT_7010_HI_ALT  "FT-7010 HI ALERT BIT" %
%   B9:0/15  FT_7010_HIHI_ALT  "FT-7010 HIHI ALERT BIT" %
%   B9:2/9  FT_7000_LOLO_ALT  "FT-7000 LOLO ALERT BIT" %
%   B9:2/11  FT_7000_LO_ALT  "FT-7000 LO ALERT BIT" %
%   B9:2/13  FT_7000_HI_ALT  "FT-7000 HI ALERT BIT" %
%   B9:2/15  FT_7000_HIHI_ALT  "FT-7000 HIHI ALERT BIT" %
%   B9:3/1  FT_7005_LOLO_ALT  "FT-7005 LOLO ALERT BIT" %
%   B9:3/3  FT_7005_LO_ALT  "FT-7005 LO ALERT BIT" %
%   B9:3/5  FT_7005_HI_ALT  "FT-7005 HI ALERT BIT" %
%   B9:3/7  FT_7005_HIHI_ALT  "FT-7005 HIHI ALERT BIT" %
%   B9:3/9  FT_7008_LOLO_ALT  "FT-7008 LOLO ALERT BIT" %
%   B9:3/11  FT_7008_LO_ALT  "FT-7008 LO ALERT BIT" %
%   B9:3/13  FT_7008_HI_ALT  "FT-7008 HI ALERT BIT" %
%   B9:3/15  FT_7008_HIHI_ALT  "FT-7008 HIHI ALERT BIT" %
%   B9:4/1  FT_7025_LOLO_ALT  "FT-7025 LOLO ALERT BIT" %
%   B9:4/3  FT_7025_LO_ALT  "FT-7025 LO ALERT BIT" %
%   B9:4/5  FT_7025_HI_ALT  "FT-7025 HI ALERT BIT" %
%   B9:4/7  FT_7025_HIHI_ALT  "FT-7025 HIHI ALERT BIT" %
%   B9:4/9  FT_7050_LOLO_ALT  "FT-7050 LOLO ALERT BIT" %
%   B9:4/11  FT_7050_LO_ALT  "FT-7050 LO ALERT BIT" %
%   B9:4/13  FT_7050_HI_ALT  "FT-7050 HI ALERT BIT" %
%   B9:4/15  FT_7050_HIHI_ALT  "FT-7050 HIHI ALERT BIT" %
%   B9:7/1  FT_7030_LOLO_ALT  "FT-7030 LOLO ALERT BIT" %
%   B9:7/3  FT_7030_LO_ALT  "FT-7030 LO ALERT BIT" %
%   B9:7/5  FT_7030_HI_ALT  "FT-7030 HI ALERT BIT" %
%   B9:7/7  FT_7030_HIHI_ALT  "FT-7030 HIHI ALERT BIT" %
%   B9:7/9  FT_7040_LOLO_ALT  "FT-7040 LOLO ALERT BIT" %
%   B9:7/11  FT_7040_LO_ALT  "FT-7040 LO ALERT BIT" %
%   B9:7/13  FT_7040_HI_ALT  "FT-7040 HI ALERT BIT" %
%   B9:7/15  FT_7040_HIHI_ALT  "FT-7040 HIHI ALERT BIT" %
%   B9:11/9  FT_7095_LOLO_ALT  "FT-7095 LOLO ALERT BIT" %
%   B9:11/11  FT_7095_LO_ALT  "FT-7095 LO ALERT BIT" %
%   B9:11/13  FT_7095_HI_ALT  "FT-7095 HI ALERT BIT" %
%   B9:11/15  FT_7095_HIHI_ALT  "FT-7095 HIHI ALERT BIT" %
%   B9:12/1  FT_7110_LOLO_ALT  "FT-7110 LOLO ALERT BIT" %
%   B9:12/3  FT_7110_LO_ALT  "FT-7110 LO ALERT BIT" %
%   B9:12/5  FT_7110_HI_ALT  "FT-7110 HI ALERT BIT" %
%   B9:12/7  FT_7110_HIHI_ALT  "FT-7110 HIHI ALERT BIT" %
%   B9:12/9  FT_7130_LOLO_ALT  "FT-7130 LOLO ALERT BIT" %
%   B9:12/11  FT_7130_LO_ALT  "FT-7130 LO ALERT BIT" %
%   B9:12/13  FT_7130_HI_ALT  "FT-7130 HI ALERT BIT" %
%   B9:12/15  FT_7130_HIHI_ALT  "FT-7130 HIHI ALERT BIT" %
%   B9:13/1  FT_7132_LOLO_ALT  "FT-7132 LOLO ALERT BIT" %
%   B9:13/3  FT_7132_LO_ALT  "FT-7132 LO ALERT BIT" %
%   B9:13/5  FT_7132_HI_ALT  "FT-7132 HI ALERT BIT" %
%   B9:13/7  FT_7132_HIHI_ALT  "FT-7132 HIHI ALERT BIT" %
%   B9:13/9  FT_7145_LOLO_ALT  "FT-7145 LOLO ALERT BIT" %
%   B9:13/11  FT_7145_LO_ALT  "FT-7145 LO ALERT BIT" %
%   B9:13/13  FT_7145_HI_ALT  "FT-7145 HI ALERT BIT" %
%   B9:13/15  FT_7145_HIHI_ALT  "FT-7145 HIHI ALERT BIT" %
%   B9:18/1  FT_7120_LOLO_ALT  "FT-7120 LOLO ALERT BIT" %
%   B9:18/3  FT_7120_LO_ALT  "FT-7120 LO ALERT BIT" %
%   B9:18/5  FT_7120_HI_ALT  "FT-7120 HI ALERT BIT" %
%   B9:18/7  FT_7120_HIHI_ALT  "FT-7120 HIHI ALERT BIT" %
%   B9:18/9  FT_7140_LOLO_ALT  "FT-7140 LOLO ALERT BIT" %
%   B9:18/11  FT_7140_LO_ALT  "FT-7140 LO ALERT BIT" %
%   B9:18/13  FT_7140_HI_ALT  "FT-7140 HI ALERT BIT" %
%   B9:18/15  FT_7140_HIHI_ALT  "FT-7140 HIHI ALERT BIT" %
%   B9:8/1  FT_7052_LOLO_ALT  "FT-7052 LOLO ALERT BIT" %
%   B9:8/3  FT_7052_LO_ALT  "FT-7052 LO ALERT BIT" %
%   B9:8/5  FT_7052_HI_ALT  "FT-7052 HI ALERT BIT" %
%   B9:8/7  FT_7052_HIHI_ALT  "FT-7052 HIHI ALERT BIT" %
%   B9:31/12  FT_ALERT  "FT ALERT" %

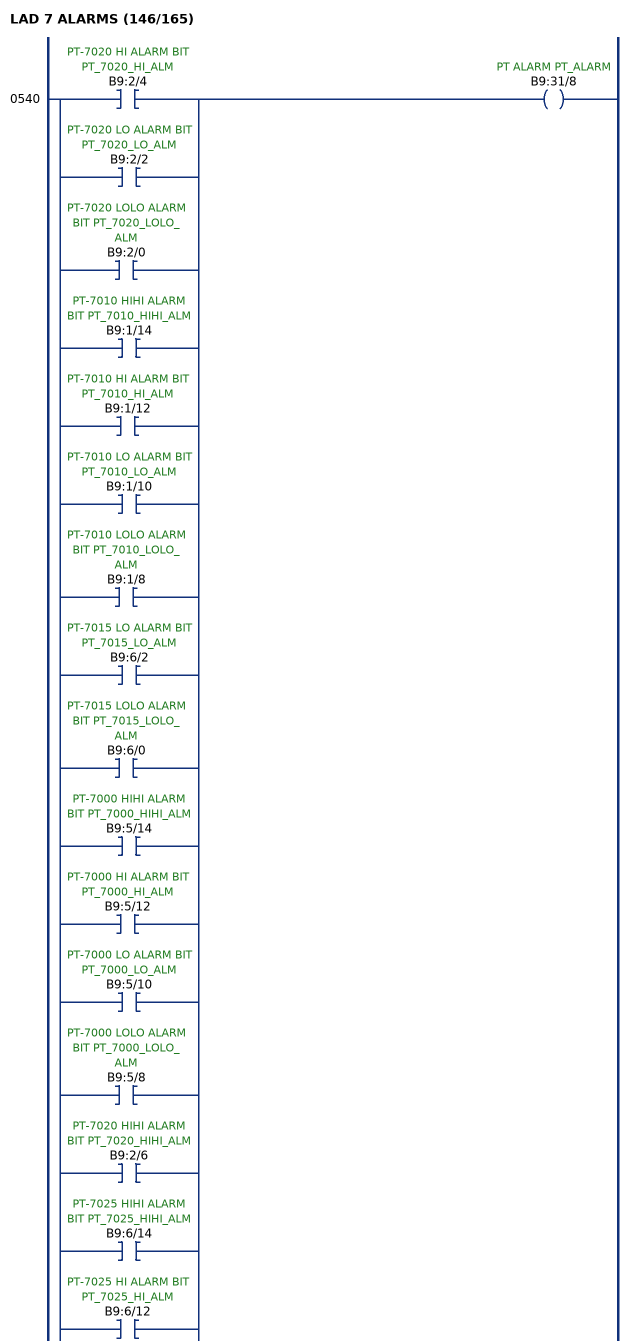

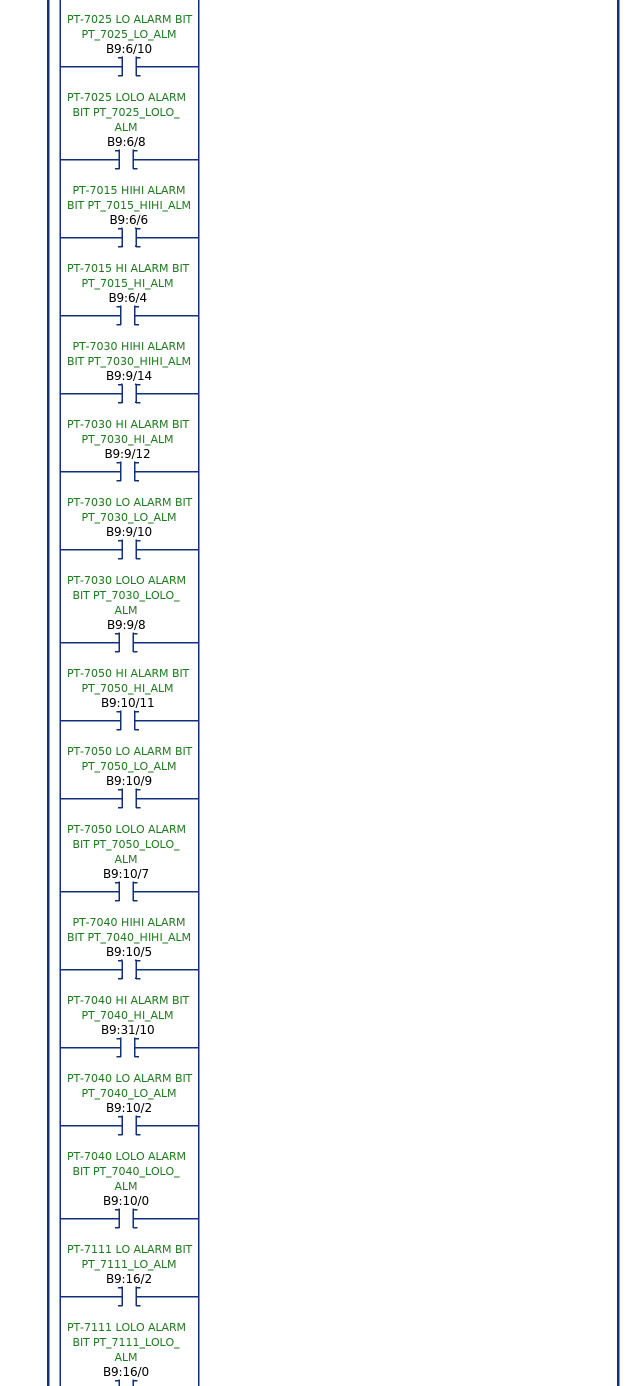

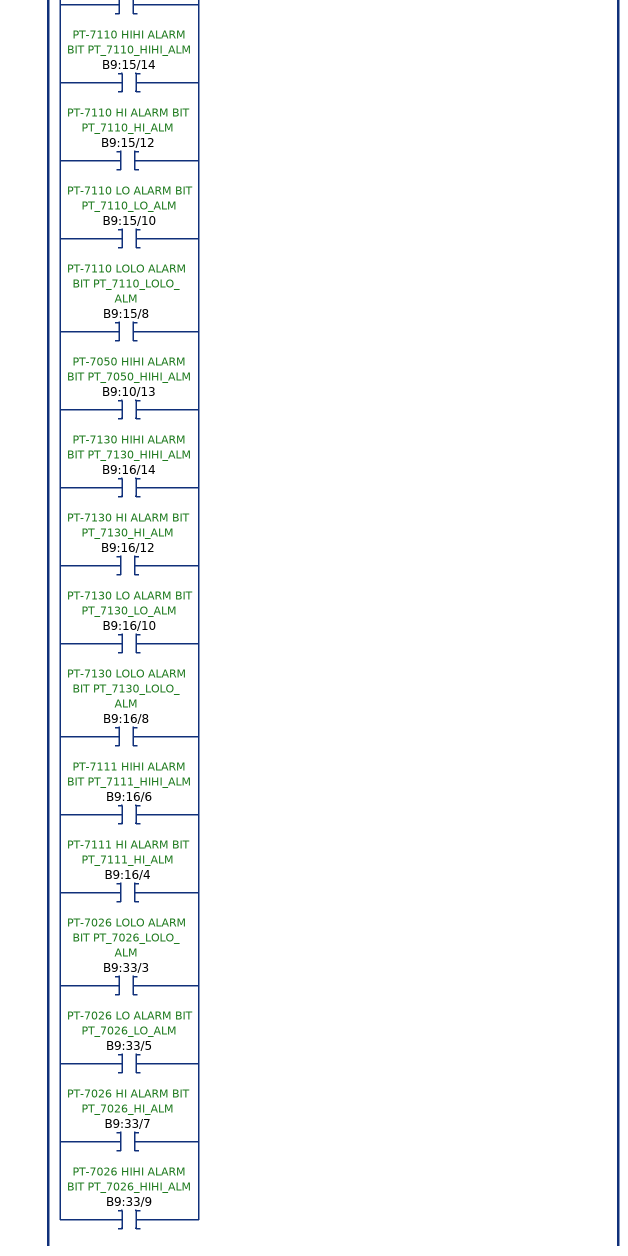
% Rung: 540 %
SOR BST XIC B9:2/4 NXB XIC B9:2/2 NXB XIC B9:2/0 NXB XIC B9:1/14 NXB XIC B9:1/12 NXB XIC B9:1/10 NXB XIC B9:1/8 NXB XIC B9:6/2 NXB XIC B9:6/0 NXB XIC B9:5/14 NXB XIC B9:5/12 NXB XIC B9:5/10 NXB XIC B9:5/8 NXB XIC B9:2/6 NXB XIC B9:6/14 NXB XIC B9:6/12 NXB XIC B9:6/10 NXB XIC B9:6/8 NXB XIC B9:6/6 NXB XIC B9:6/4 NXB XIC B9:9/14 NXB XIC B9:9/12 NXB XIC B9:9/10 NXB XIC B9:9/8 NXB XIC B9:10/11 NXB XIC B9:10/9 NXB XIC B9:10/7 NXB XIC B9:10/5 NXB XIC B9:31/10 NXB XIC B9:10/2 NXB XIC B9:10/0 NXB XIC B9:16/2 NXB XIC B9:16/0 NXB XIC B9:15/14 NXB XIC B9:15/12 NXB XIC B9:15/10 NXB XIC B9:15/8 NXB XIC B9:10/13 NXB XIC B9:16/14 NXB XIC B9:16/12 NXB XIC B9:16/10 NXB XIC B9:16/8 NXB XIC B9:16/6 NXB XIC B9:16/4 NXB XIC B9:33/3 NXB XIC B9:33/5 NXB XIC B9:33/7 NXB XIC B9:33/9 BND OTE B9:31/8 EOR
%   B9:2/4  PT_7020_HI_ALM  "PT-7020 HI ALARM BIT" %
%   B9:2/2  PT_7020_LO_ALM  "PT-7020 LO ALARM BIT" %
%   B9:2/0  PT_7020_LOLO_ALM  "PT-7020 LOLO ALARM BIT" %
%   B9:1/14  PT_7010_HIHI_ALM  "PT-7010 HIHI ALARM BIT" %
%   B9:1/12  PT_7010_HI_ALM  "PT-7010 HI ALARM BIT" %
%   B9:1/10  PT_7010_LO_ALM  "PT-7010 LO ALARM BIT" %
%   B9:1/8  PT_7010_LOLO_ALM  "PT-7010 LOLO ALARM BIT" %
%   B9:6/2  PT_7015_LO_ALM  "PT-7015 LO ALARM BIT" %
%   B9:6/0  PT_7015_LOLO_ALM  "PT-7015 LOLO ALARM BIT" %
%   B9:5/14  PT_7000_HIHI_ALM  "PT-7000 HIHI ALARM BIT" %
%   B9:5/12  PT_7000_HI_ALM  "PT-7000 HI ALARM BIT" %
%   B9:5/10  PT_7000_LO_ALM  "PT-7000 LO ALARM BIT" %
%   B9:5/8  PT_7000_LOLO_ALM  "PT-7000 LOLO ALARM BIT" %
%   B9:2/6  PT_7020_HIHI_ALM  "PT-7020 HIHI ALARM BIT" %
%   B9:6/14  PT_7025_HIHI_ALM  "PT-7025 HIHI ALARM BIT" %
%   B9:6/12  PT_7025_HI_ALM  "PT-7025 HI ALARM BIT" %
%   B9:6/10  PT_7025_LO_ALM  "PT-7025 LO ALARM BIT" %
%   B9:6/8  PT_7025_LOLO_ALM  "PT-7025 LOLO ALARM BIT" %
%   B9:6/6  PT_7015_HIHI_ALM  "PT-7015 HIHI ALARM BIT" %
%   B9:6/4  PT_7015_HI_ALM  "PT-7015 HI ALARM BIT" %
%   B9:9/14  PT_7030_HIHI_ALM  "PT-7030 HIHI ALARM BIT" %
%   B9:9/12  PT_7030_HI_ALM  "PT-7030 HI ALARM BIT" %
%   B9:9/10  PT_7030_LO_ALM  "PT-7030 LO ALARM BIT" %
%   B9:9/8  PT_7030_LOLO_ALM  "PT-7030 LOLO ALARM BIT" %
%   B9:10/11  PT_7050_HI_ALM  "PT-7050 HI ALARM BIT" %
%   B9:10/9  PT_7050_LO_ALM  "PT-7050 LO ALARM BIT" %
%   B9:10/7  PT_7050_LOLO_ALM  "PT-7050 LOLO ALARM BIT" %
%   B9:10/5  PT_7040_HIHI_ALM  "PT-7040 HIHI ALARM BIT" %
%   B9:31/10  PT_7040_HI_ALM  "PT-7040 HI ALARM BIT" %
%   B9:10/2  PT_7040_LO_ALM  "PT-7040 LO ALARM BIT" %
%   B9:10/0  PT_7040_LOLO_ALM  "PT-7040 LOLO ALARM BIT" %
%   B9:16/2  PT_7111_LO_ALM  "PT-7111 LO ALARM BIT" %
%   B9:16/0  PT_7111_LOLO_ALM  "PT-7111 LOLO ALARM BIT" %
%   B9:15/14  PT_7110_HIHI_ALM  "PT-7110 HIHI ALARM BIT" %
%   B9:15/12  PT_7110_HI_ALM  "PT-7110 HI ALARM BIT" %
%   B9:15/10  PT_7110_LO_ALM  "PT-7110 LO ALARM BIT" %
%   B9:15/8  PT_7110_LOLO_ALM  "PT-7110 LOLO ALARM BIT" %
%   B9:10/13  PT_7050_HIHI_ALM  "PT-7050 HIHI ALARM BIT" %
%   B9:16/14  PT_7130_HIHI_ALM  "PT-7130 HIHI ALARM BIT" %
%   B9:16/12  PT_7130_HI_ALM  "PT-7130 HI ALARM BIT" %
%   B9:16/10  PT_7130_LO_ALM  "PT-7130 LO ALARM BIT" %
%   B9:16/8  PT_7130_LOLO_ALM  "PT-7130 LOLO ALARM BIT" %
%   B9:16/6  PT_7111_HIHI_ALM  "PT-7111 HIHI ALARM BIT" %
%   B9:16/4  PT_7111_HI_ALM  "PT-7111 HI ALARM BIT" %
%   B9:33/3  PT_7026_LOLO_ALM  "PT-7026 LOLO ALARM BIT" %
%   B9:33/5  PT_7026_LO_ALM  "PT-7026 LO ALARM BIT" %
%   B9:33/7  PT_7026_HI_ALM  "PT-7026 HI ALARM BIT" %
%   B9:33/9  PT_7026_HIHI_ALM  "PT-7026 HIHI ALARM BIT" %
%   B9:31/8  PT_ALARM  "PT ALARM" %

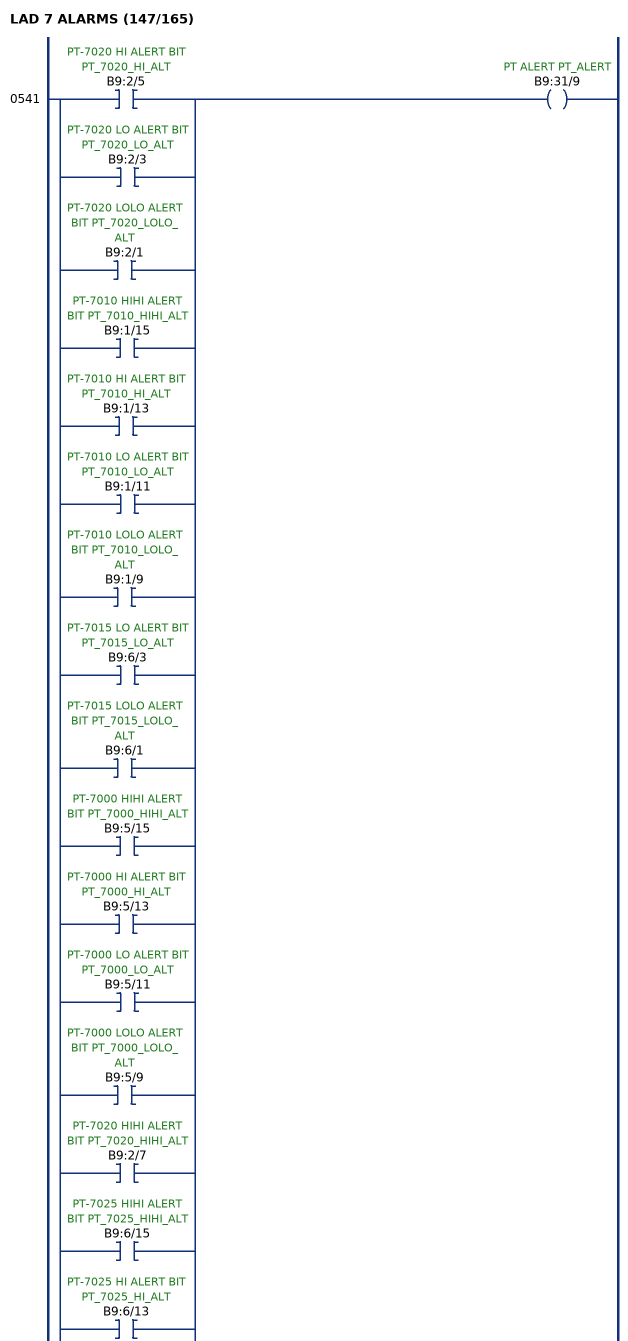

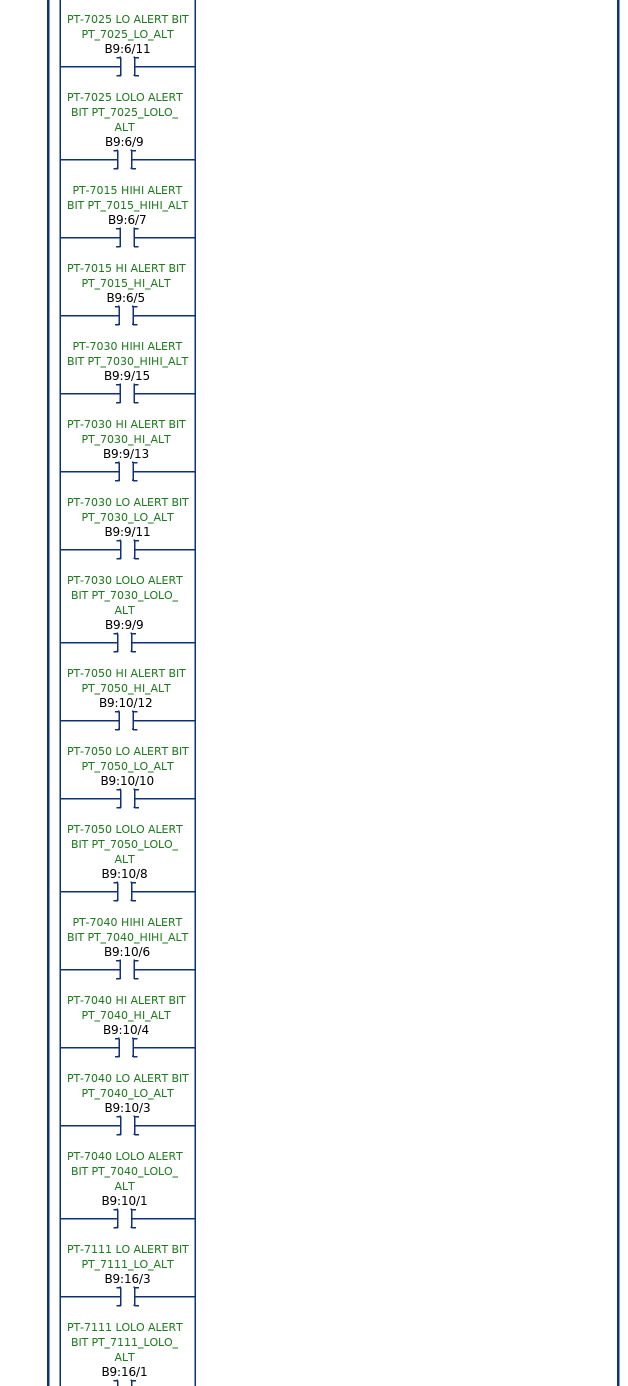

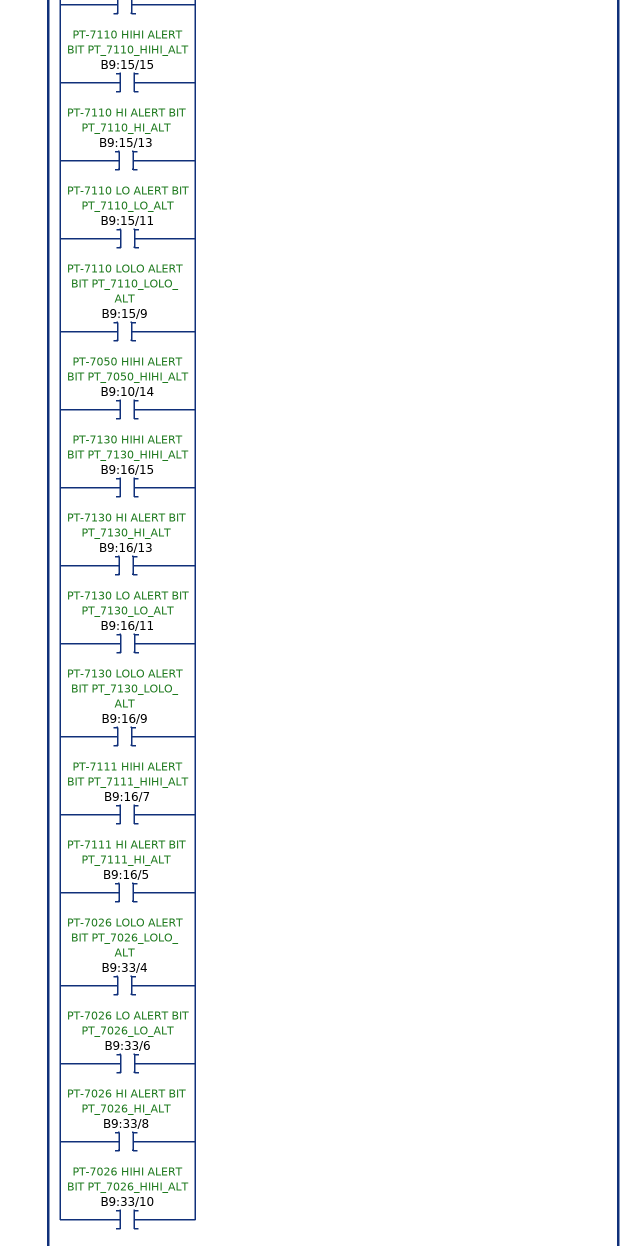
% Rung: 541 %
SOR BST XIC B9:2/5 NXB XIC B9:2/3 NXB XIC B9:2/1 NXB XIC B9:1/15 NXB XIC B9:1/13 NXB XIC B9:1/11 NXB XIC B9:1/9 NXB XIC B9:6/3 NXB XIC B9:6/1 NXB XIC B9:5/15 NXB XIC B9:5/13 NXB XIC B9:5/11 NXB XIC B9:5/9 NXB XIC B9:2/7 NXB XIC B9:6/15 NXB XIC B9:6/13 NXB XIC B9:6/11 NXB XIC B9:6/9 NXB XIC B9:6/7 NXB XIC B9:6/5 NXB XIC B9:9/15 NXB XIC B9:9/13 NXB XIC B9:9/11 NXB XIC B9:9/9 NXB XIC B9:10/12 NXB XIC B9:10/10 NXB XIC B9:10/8 NXB XIC B9:10/6 NXB XIC B9:10/4 NXB XIC B9:10/3 NXB XIC B9:10/1 NXB XIC B9:16/3 NXB XIC B9:16/1 NXB XIC B9:15/15 NXB XIC B9:15/13 NXB XIC B9:15/11 NXB XIC B9:15/9 NXB XIC B9:10/14 NXB XIC B9:16/15 NXB XIC B9:16/13 NXB XIC B9:16/11 NXB XIC B9:16/9 NXB XIC B9:16/7 NXB XIC B9:16/5 NXB XIC B9:33/4 NXB XIC B9:33/6 NXB XIC B9:33/8 NXB XIC B9:33/10 BND OTE B9:31/9 EOR
%   B9:2/5  PT_7020_HI_ALT  "PT-7020 HI ALERT BIT" %
%   B9:2/3  PT_7020_LO_ALT  "PT-7020 LO ALERT BIT" %
%   B9:2/1  PT_7020_LOLO_ALT  "PT-7020 LOLO ALERT BIT" %
%   B9:1/15  PT_7010_HIHI_ALT  "PT-7010 HIHI ALERT BIT" %
%   B9:1/13  PT_7010_HI_ALT  "PT-7010 HI ALERT BIT" %
%   B9:1/11  PT_7010_LO_ALT  "PT-7010 LO ALERT BIT" %
%   B9:1/9  PT_7010_LOLO_ALT  "PT-7010 LOLO ALERT BIT" %
%   B9:6/3  PT_7015_LO_ALT  "PT-7015 LO ALERT BIT" %
%   B9:6/1  PT_7015_LOLO_ALT  "PT-7015 LOLO ALERT BIT" %
%   B9:5/15  PT_7000_HIHI_ALT  "PT-7000 HIHI ALERT BIT" %
%   B9:5/13  PT_7000_HI_ALT  "PT-7000 HI ALERT BIT" %
%   B9:5/11  PT_7000_LO_ALT  "PT-7000 LO ALERT BIT" %
%   B9:5/9  PT_7000_LOLO_ALT  "PT-7000 LOLO ALERT BIT" %
%   B9:2/7  PT_7020_HIHI_ALT  "PT-7020 HIHI ALERT BIT" %
%   B9:6/15  PT_7025_HIHI_ALT  "PT-7025 HIHI ALERT BIT" %
%   B9:6/13  PT_7025_HI_ALT  "PT-7025 HI ALERT BIT" %
%   B9:6/11  PT_7025_LO_ALT  "PT-7025 LO ALERT BIT" %
%   B9:6/9  PT_7025_LOLO_ALT  "PT-7025 LOLO ALERT BIT" %
%   B9:6/7  PT_7015_HIHI_ALT  "PT-7015 HIHI ALERT BIT" %
%   B9:6/5  PT_7015_HI_ALT  "PT-7015 HI ALERT BIT" %
%   B9:9/15  PT_7030_HIHI_ALT  "PT-7030 HIHI ALERT BIT" %
%   B9:9/13  PT_7030_HI_ALT  "PT-7030 HI ALERT BIT" %
%   B9:9/11  PT_7030_LO_ALT  "PT-7030 LO ALERT BIT" %
%   B9:9/9  PT_7030_LOLO_ALT  "PT-7030 LOLO ALERT BIT" %
%   B9:10/12  PT_7050_HI_ALT  "PT-7050 HI ALERT BIT" %
%   B9:10/10  PT_7050_LO_ALT  "PT-7050 LO ALERT BIT" %
%   B9:10/8  PT_7050_LOLO_ALT  "PT-7050 LOLO ALERT BIT" %
%   B9:10/6  PT_7040_HIHI_ALT  "PT-7040 HIHI ALERT BIT" %
%   B9:10/4  PT_7040_HI_ALT  "PT-7040 HI ALERT BIT" %
%   B9:10/3  PT_7040_LO_ALT  "PT-7040 LO ALERT BIT" %
%   B9:10/1  PT_7040_LOLO_ALT  "PT-7040 LOLO ALERT BIT" %
%   B9:16/3  PT_7111_LO_ALT  "PT-7111 LO ALERT BIT" %
%   B9:16/1  PT_7111_LOLO_ALT  "PT-7111 LOLO ALERT BIT" %
%   B9:15/15  PT_7110_HIHI_ALT  "PT-7110 HIHI ALERT BIT" %
%   B9:15/13  PT_7110_HI_ALT  "PT-7110 HI ALERT BIT" %
%   B9:15/11  PT_7110_LO_ALT  "PT-7110 LO ALERT BIT" %
%   B9:15/9  PT_7110_LOLO_ALT  "PT-7110 LOLO ALERT BIT" %
%   B9:10/14  PT_7050_HIHI_ALT  "PT-7050 HIHI ALERT BIT" %
%   B9:16/15  PT_7130_HIHI_ALT  "PT-7130 HIHI ALERT BIT" %
%   B9:16/13  PT_7130_HI_ALT  "PT-7130 HI ALERT BIT" %
%   B9:16/11  PT_7130_LO_ALT  "PT-7130 LO ALERT BIT" %
%   B9:16/9  PT_7130_LOLO_ALT  "PT-7130 LOLO ALERT BIT" %
%   B9:16/7  PT_7111_HIHI_ALT  "PT-7111 HIHI ALERT BIT" %
%   B9:16/5  PT_7111_HI_ALT  "PT-7111 HI ALERT BIT" %
%   B9:33/4  PT_7026_LOLO_ALT  "PT-7026 LOLO ALERT BIT" %
%   B9:33/6  PT_7026_LO_ALT  "PT-7026 LO ALERT BIT" %
%   B9:33/8  PT_7026_HI_ALT  "PT-7026 HI ALERT BIT" %
%   B9:33/10  PT_7026_HIHI_ALT  "PT-7026 HIHI ALERT BIT" %
%   B9:31/9  PT_ALERT  "PT ALERT" %

